	STARTING:
		FOR i := 1 TO fbCurrentSequence.stepsTotal() BY 1 DO
			Steps := fbCurrentSequence.steps();
			Steps[i].Device^.enable();
		END_FOR
		
	
		nCurrentStepPreviousCycle := nCurrentStep;
		
		// Attempt next step execution for a wait for action step
		IF Steps[nCurrentStep].WaitForAction THEN
			IF(executeStep(fbCurrentSequence.step(nCurrentStep)) AND nCurrentStep <> fbCurrentSequence.stepsTotal()) THEN
				nCurrentStep := nCurrentStep + 1;	
			END_IF
		END_IF
		
		// Attempt next step execution for a non wait for action step
		IF NOT Steps[nCurrentStep].WaitForAction THEN
			fbCurrentSequence.step(nCurrentStep)^.Device^.setCommand(StateTarget := fbCurrentSequence.step(nCurrentStep)^.Command);
			nCurrentStep := nCurrentStep + 1;	
		END_IF
		
		
		// Check which sequence step we are up to, set the currentStep indicator to +1 of where we are
		// Interlocks / permissives can cause us to go backwards in steps, therefore we must do this check
		
		IF NOT fbCurrentSequence.getSeqType() THEN // only do this check if it is a flooding sequence
			checkCurrentStep();	
			IF nCurrentStep < nCurrentStepPreviousCycle THEN  // an interlock has caused the program to roll back in sequence (interlock etc.) - stay in PAUSE state and wait for user acknowledgement
				eSMState := HOLD;
			END_IF
		END_IF
			
		eState := E_SequenceState.STARTING;
	
		
		
		
	RUNNING:


// Sequence is running - just need to check that we are still running, if not, we go to paused
		nCurrentStepPreviousCycle := nCurrentStep;
		
		IF NOT fbCurrentSequence.getSeqType() THEN // only do this check if it is a flooding sequence
			checkCurrentStep();
			IF nCurrentStep < fbCurrentSequence.stepsTotal() THEN  // something has forced us out of the running state, go to paused and wait for operator to acknowledge
				eSMState := HOLD;
			END_IF
		END_IF
		
		IF NOT (fbCurrentSequence.getSeqType()) THEN // the sequence is a floop type sequence
			eState := E_SequenceState.RUN;
		ELSIF NOT (fbCurrentSequence.step(StepNum := nCurrentStep)^.Device^.getState() = fbCurrentSequence.stepCommand(StepNumber := nCurrentStep)) THEN
			eSMState := STARTING;
		END_IF
		
		
	HOLD:
		// Do not progress the sequence until the operator has acknowledged that something went wrong
		IF bPauseAcknowledged THEN
			eSMState := STARTING;
			bPauseAcknowledged := FALSE;
		END_IF
		
		eState := E_SequenceState.HOLD;
		
	COMPLETE:
		eState := E_SequenceState.COMPLETE;
		
		
END_CASE

METHOD acknowledgePause : BOOL
VAR_INPUT
END_VAR
bPauseAcknowledged := TRUE;
END_METHOD

METHOD addSequence : BOOL
VAR_INPUT
	Sequence: FB_SequenceBase;
END_VAR
aSequences[nNumberSequences + 1] := Sequence;
nNumberSequences := nNumberSequences + 1;
END_METHOD

METHOD checkCurrentStep : BOOL
VAR_INPUT
END_VAR

VAR
	currentState: E_DeviceState;
	targetState: E_DeviceState;
END_VAR
nCurrentStepCheck := 1;

WHILE nCurrentStepCheck < (fbCurrentSequence.stepsTotal() + 1) DO
	
	currentState := fbCurrentSequence.stepState(nCurrentStepCheck);
	targetState := fbCurrentSequence.stepCommand(nCurrentStepCheck);

	IF currentState = targetState THEN
		nCurrentStepCheck := nCurrentStepCheck + 1;
	ELSE
		nCurrentStep := nCurrentStepCheck; // step check reveals we are here
		nCurrentStepCheck := fbCurrentSequence.stepsTotal() + 1; // terminate loop as the checking is finished
	END_IF
END_WHILE
END_METHOD

METHOD executeStep : BOOL
VAR_INPUT
	stSequenceStep: POINTER TO ST_SequenceStep;
END_VAR

VAR
	(*eCheckState: E_DeviceState;
	eCheckStateAlternative: E_DeviceState;
	eCheckStateAlternative2: E_DeviceState;
	eCheckCommand: E_DeviceState;
	fbDevice: POINTER TO FB_BaseDevice;
	*)
END_VAR
executeStep := FALSE;


IF fbCurrentSequence.step(StepNum := nCurrentStep)^.Device^.getState()  
	= fbCurrentSequence.stepCommand(StepNumber := nCurrentStep)
	AND fbTONstep.Q THEN  
	
	IF (nCurrentStep = fbCurrentSequence.stepsTotal() AND fbCurrentSequence.getSeqType()) THEN
		eSMState := COMPLETE;
	ELSIF (nCurrentStep = fbCurrentSequence.stepsTotal() AND (NOT fbCurrentSequence.getSeqType())) THEN
		eSMState := RUNNING;
	END_IF
	//fbTONdelay.IN := FALSE;
	fbTONdelay(IN:= TRUE, PT := stSequenceStep^.DelayUntilNextStep); 
	
	executeStep := TRUE; // indicate that the step was sucessful
	
	
ELSIF (fbCurrentSequence.step(StepNum := nCurrentStep)^.Device^.isEnabled() ) AND 
		(NOT (fbCurrentSequence.step(StepNum := nCurrentStep)^.Device^.getMode() = E_DeviceMode.MANUAL)) AND
		fbTONdelay.Q THEN 
	//AND fbTONdelay.Q THEN
		
		//fbTONdelay.IN := FALSE; 		
		fbTONdelay.IN := FALSE;
		fbTONstep(IN:= TRUE, PT := stSequenceStep^.StepMinDuration);		
		stSequenceStep^.Device^.setCommand(StateTarget := stSequenceStep^.Command); // set the target state 

END_IF

(*
IF fbCurrentSequence.step(StepNum := nCurrentStep)^.Device^.getState()  
	= fbCurrentSequence.step(StepNum := nCurrentStep)^.Device^.getCommand() 
	AND fbTONstep.Q THEN  *)
END_METHOD

METHOD getCurrentSeq_FB : POINTER TO FB_SequenceBase
VAR_INPUT
END_VAR
getCurrentSeq_FB := ADR(fbCurrentSequence);
END_METHOD

METHOD getCurrentSeq_ID : INT
VAR_INPUT
END_VAR
getCurrentSeq_ID := nCurrentSequence;
END_METHOD

METHOD getState : E_SequenceState
VAR_INPUT
END_VAR
getState := eState;
END_METHOD

METHOD initSequence : BOOL
VAR_INPUT
END_VAR
// We want to iterate through all of the components in a sequence and enable them.
// We also want to disable any other device (provided it is not in manual)
END_METHOD

METHOD pauseSequence : BOOL
VAR_INPUT
END_VAR
eSMState := HOLD;
END_METHOD

METHOD selectSequence : BOOL
VAR_INPUT
	Sequence: INT;
END_VAR
fbCurrentSequence := aSequences[Sequence];
nCurrentSequence := Sequence;
END_METHOD

METHOD startSequence : BOOL
VAR_INPUT
END_VAR
VAR

END_VAR
eSMState := STARTING;

FOR i := 1 TO fbCurrentSequence.stepsTotal() BY 1 DO
	Steps := fbCurrentSequence.steps();
	Steps[i].Device^.enable();
END_FOR

nCurrentStep := 1;
nCurrentStepPreviousCycle := 1;
//nCurrentSequence := 1;
nCurrentStepCheck := 1; 

fbTONdelay(PT := T#1s, IN := TRUE);
END_METHOD

METHOD stopSequence : BOOL
VAR_INPUT
END_VAR
eSMState := STOPPED;


FOR i := 1 TO fbCurrentSequence.stepsTotal() BY 1 DO
	Steps := fbCurrentSequence.steps();
	Steps[i].Device^.disable();
END_FOR
END_METHOD

END_FUNCTION_BLOCK

// ---- POUs/05 Sequences/FB_SequenceBase.TcPOU
(*
		This function block serves as a template for all machine sequences
		Each sequence step is a structure (ST_SequenceStep) which is defined in the FB_Init
		method of machine sequence function blocks that extend this FB.
		After the steps are defined, the STs are packed into the array 'aSequenceSteps'
		which is used by the Sequence Manager whom iterates over this array to co-ordinate 
		the execution of steps and/or detection of where sequences are interruped by interlock
		conditions
*)

FUNCTION_BLOCK FB_SequenceBase

(*
VAR_IN_OUT
	{attribute 'OPC.UA.DA' := '0'} 
	devices: ST_DMComponents;
END_VAR
*)


VAR
	sSequenceName: STRING;
	sSequenceDescription: STRING(245);
	nNumberSequenceSteps: INT;
	
	
	bSequentional_1_Flood_0: BOOL := FALSE; // default to flood and set to TRUE using setSequential() method
	
	aSequenceSteps: ARRAY[1..20] OF ST_SequenceStep;
	//aSequenceSteps: ARRAY[1..20] OF ST_SequenceStep;
	{attribute 'OPC.UA.DA' := '0'} 
	Step1: ST_SequenceStep;
	{attribute 'OPC.UA.DA' := '0'} 
	Step2: ST_SequenceStep;
	{attribute 'OPC.UA.DA' := '0'} 
	Step3: ST_SequenceStep;
	{attribute 'OPC.UA.DA' := '0'} 
	Step4: ST_SequenceStep;
	{attribute 'OPC.UA.DA' := '0'} 
	Step5: ST_SequenceStep;
	{attribute 'OPC.UA.DA' := '0'} 
	Step6: ST_SequenceStep;
	{attribute 'OPC.UA.DA' := '0'} 
	Step7: ST_SequenceStep;
	{attribute 'OPC.UA.DA' := '0'} 
	Step8: ST_SequenceStep;
	{attribute 'OPC.UA.DA' := '0'} 
	Step9: ST_SequenceStep;
	{attribute 'OPC.UA.DA' := '0'} 
	Step10: ST_SequenceStep;
	{attribute 'OPC.UA.DA' := '0'} 
	Step11: ST_SequenceStep;
	{attribute 'OPC.UA.DA' := '0'} 
	Step12: ST_SequenceStep;
	{attribute 'OPC.UA.DA' := '0'} 
	Step13: ST_SequenceStep;
	{attribute 'OPC.UA.DA' := '0'} 
	Step14: ST_SequenceStep;
	{attribute 'OPC.UA.DA' := '0'} 
	Step15: ST_SequenceStep;
	{attribute 'OPC.UA.DA' := '0'} 
	Step16: ST_SequenceStep;
	{attribute 'OPC.UA.DA' := '0'} 
	Step17: ST_SequenceStep;
	{attribute 'OPC.UA.DA' := '0'} 
	Step18: ST_SequenceStep;
	{attribute 'OPC.UA.DA' := '0'} 
	Step19: ST_SequenceStep;
	{attribute 'OPC.UA.DA' := '0'} 
	Step20: ST_SequenceStep;
	{attribute 'OPC.UA.DA' := '0'} 
	Step21: ST_SequenceStep;
	{attribute 'OPC.UA.DA' := '0'} 
	Step22: ST_SequenceStep;
	{attribute 'OPC.UA.DA' := '0'} 
	Step23: ST_SequenceStep;
	{attribute 'OPC.UA.DA' := '0'} 
	Step24: ST_SequenceStep;
	{attribute 'OPC.UA.DA' := '0'} 
	Step25: ST_SequenceStep;
	{attribute 'OPC.UA.DA' := '0'} 
	Step26: ST_SequenceStep;
	{attribute 'OPC.UA.DA' := '0'} 
	Step27: ST_SequenceStep;
	{attribute 'OPC.UA.DA' := '0'} 
	Step28: ST_SequenceStep;
END_VAR

(*
	Use the text below in the FBs that extend this to build the sequence
	
			Step1.Component := devices.
			Step1.Command := E_DeviceState.
			Step1.StepMinDuration := T#5S; 
			Step1.DelayUntilNextStep := T#5S;
			Step1.WaitForAction := TRUE;
			aSequenceSteps[1] :=   Step1;
			
			
			Step2.Component := devices.
			Step2.Command := E_DeviceState.
			Step2.StepMinDuration := T#5S; 
			Step2.DelayUntilNextStep := T#5S;
			Step2.WaitForAction := TRUE;
			aSequenceSteps[2] :=   Step2;
			
			
			Step3.Component := devices.
			Step3.Command := E_DeviceState.
			Step3.StepMinDuration := T#5S; 
			Step3.DelayUntilNextStep := T#5S;
			Step3.WaitForAction := TRUE;
			aSequenceSteps[3] :=   Step3;
			
			
			Step4.Component := devices.
			Step4.Command := E_DeviceState.
			Step4.StepMinDuration := T#5S; 
			Step4.DelayUntilNextStep := T#5S;
			Step4.WaitForAction := TRUE;
			aSequenceSteps[4] :=   Step4;
			
			
			Step5.Component := devices.
			Step5.Command := E_DeviceState.
			Step5.StepMinDuration := T#5S; 
			Step5.DelayUntilNextStep := T#5S;
			Step5.WaitForAction := TRUE;
			aSequenceSteps[5] :=   Step5;
			
			
			Step6.Component := devices.
			Step6.Command := E_DeviceState.
			Step6.StepMinDuration := T#5S; 
			Step6.DelayUntilNextStep := T#5S;
			Step6.WaitForAction := TRUE;
			aSequenceSteps[6] :=   Step6;
			
			
			Step7.Component := devices.
			Step7.Command := E_DeviceState.
			Step7.StepMinDuration := T#5S; 
			Step7.DelayUntilNextStep := T#5S;
			Step7.WaitForAction := TRUE;
			aSequenceSteps[7] :=   Step7;
			
			
			Step8.Component := devices.
			Step8.Command := E_DeviceState.
			Step8.StepMinDuration := T#5S; 
			Step8.DelayUntilNextStep := T#5S;
			Step8.WaitForAction := TRUE;
			aSequenceSteps[8] :=   Step8;
			
			
			Step9.Component := devices.
			Step9.Command := E_DeviceState.
			Step9.StepMinDuration := T#5S; 
			Step9.DelayUntilNextStep := T#5S;
			Step9.WaitForAction := TRUE;
			aSequenceSteps[9] :=   Step9;
			
			
			Step10.Component := devices.
			Step10.Command := E_DeviceState.
			Step10.StepMinDuration := T#5S; 
			Step10.DelayUntilNextStep := T#5S;
			Step10.WaitForAction := TRUE;
			aSequenceSteps[10] :=   Step10;
			
			
			Step11.Component := devices.
			Step11.Command := E_DeviceState.
			Step11.StepMinDuration := T#5S; 
			Step11.DelayUntilNextStep := T#5S;
			Step11.WaitForAction := TRUE;
			aSequenceSteps[11] :=   Step11;
			
			
			Step12.Component := devices.
			Step12.Command := E_DeviceState.
			Step12.StepMinDuration := T#5S; 
			Step12.DelayUntilNextStep := T#5S;
			Step12.WaitForAction := TRUE;
			aSequenceSteps[12] :=   Step12;
			
			
			Step13.Component := devices.
			Step13.Command := E_DeviceState.
			Step13.StepMinDuration := T#5S; 
			Step13.DelayUntilNextStep := T#5S;
			Step13.WaitForAction := TRUE;
			aSequenceSteps[13] :=   Step13;
			
			
			Step14.Component := devices.
			Step14.Command := E_DeviceState.
			Step14.StepMinDuration := T#5S; 
			Step14.DelayUntilNextStep := T#5S;
			Step14.WaitForAction := TRUE;
			aSequenceSteps[14] :=   Step14;
			
			
			Step15.Component := devices.
			Step15.Command := E_DeviceState.
			Step15.StepMinDuration := T#5S; 
			Step15.DelayUntilNextStep := T#5S;
			Step15.WaitForAction := TRUE;
			aSequenceSteps[15] :=   Step15;
			
			
			Step16.Component := devices.
			Step16.Command := E_DeviceState.
			Step16.StepMinDuration := T#5S; 
			Step16.DelayUntilNextStep := T#5S;
			Step16.WaitForAction := TRUE;
			aSequenceSteps[16] :=   Step16;
			
			
			Step17.Component := devices.
			Step17.Command := E_DeviceState.
			Step17.StepMinDuration := T#5S; 
			Step17.DelayUntilNextStep := T#5S;
			Step17.WaitForAction := TRUE;
			aSequenceSteps[17] :=   Step17;
			
			
			Step18.Component := devices.
			Step18.Command := E_DeviceState.
			Step18.StepMinDuration := T#5S; 
			Step18.DelayUntilNextStep := T#5S;
			Step18.WaitForAction := TRUE;
			aSequenceSteps[18] :=   Step18;
			
			
			Step19.Component := devices.
			Step19.Command := E_DeviceState.
			Step19.StepMinDuration := T#5S; 
			Step19.DelayUntilNextStep := T#5S;
			Step19.WaitForAction := TRUE;
			aSequenceSteps[19] :=   Step19;
			
			
			Step20.Component := devices.
			Step20.Command := E_DeviceState.
			Step20.StepMinDuration := T#5S; 
			Step20.DelayUntilNextStep := T#5S;
			Step20.WaitForAction := TRUE;
			aSequenceSteps[20] :=   Step20;



*)

METHOD getSeqType : BOOL
VAR_INPUT
END_VAR
getSeqType := bSequentional_1_Flood_0;
END_METHOD

METHOD setSeqType : BOOL
VAR_INPUT
	Sequential_1_Flood_0: BOOL;
END_VAR
bSequentional_1_Flood_0 := Sequential_1_Flood_0;
END_METHOD

METHOD step : POINTER TO ST_SequenceStep
VAR_INPUT
	StepNum: INT;
END_VAR
step := ADR(aSequenceSteps[StepNum]);
END_METHOD

METHOD stepCommand : E_DeviceState
VAR_INPUT
	StepNumber: INT;
END_VAR
stepCommand := aSequenceSteps[StepNumber].Command;
END_METHOD

METHOD steps : ARRAY[1..20] OF ST_SequenceStep
VAR_INPUT
END_VAR
steps := aSequenceSteps;
END_METHOD

METHOD stepState : E_DeviceState
VAR_INPUT
	StepNumber: INT;
END_VAR
stepState := aSequenceSteps[StepNumber].Device^.getState();
END_METHOD

METHOD stepsTotal : INT
VAR_INPUT
END_VAR
stepsTotal := nNumberSequenceSteps;
END_METHOD

METHOD updateVarIDs : BOOL
VAR
	iterator: INT;
END_VAR
FOR iterator := 1 TO nNumberSequenceSteps BY 1 DO
	aSequenceSteps[iterator].DeviceVarID := aSequenceSteps[iterator].Device^.getVarID();
END_FOR
END_METHOD

END_FUNCTION_BLOCK

// ---- POUs/00 Interfaces/FB_HandShake_TrayMovement.TcPOU
FUNCTION_BLOCK FB_HandShake_TrayMovement EXTENDS FB_BaseDevice



VAR_INPUT PERSISTENT 
	stTrayExchangeInput: ST_TrayExchangeHandshake;
END_VAR

VAR_OUTPUT PERSISTENT
	stTrayExchgangeOutput: ST_TrayExchangeHandshake;
END_VAR


VAR
	fbTON_Timer: TON;			// used to time duration from bExecuture move TRUE to both bDone booleans set to true
	{attribute 'OPC.UA.DA' := '1'} 
	tDurationMovement: TIME;	// holds the duration of the last tray movement


END_VAR

VAR PERSISTENT
	{attribute 'OPC.UA.DA' := '1'} 
	tAlarmMovement: TIME;		// user specified duration for tray movement alarm
END_VAR

fbTON_Timer(IN := (stTrayExchangeInput.eState = E_TrayExchangeState.IN_PROGRESS));

IF fbTON_Timer.Q THEN
	 aErrors[1].bEnabled 	:= TRUE;
	 aErrors[1].ePriority 	:= E_AlarmPriority.High;
	 aErrors[1].sLabel 		:= 'Tray Movement Timeout';
END_IF 

IF stTrayExchangeInput.bDoneReceiver AND stTrayExchangeInput.bDoneSender THEN
	stTrayExchangeInput.eState := E_TrayExchangeState.COMPLETED;
END_IF

IF stTrayExchangeInput.eState = E_TrayExchangeState.IN_PROGRESS THEN
	stTrayExchangeInput.stTrayOutgoing := stTrayExchangeInput.stTrayIncoming;
END_IF


stTrayExchgangeOutput := stTrayExchangeInput;

END_FUNCTION_BLOCK

// ---- POUs/LFT/FB_Lift.TcPOU
FUNCTION_BLOCK FB_Lift EXTENDS FB_BaseDevice

VAR
	fbServo: FB_SEW_MovidriveB;
END_VAR

VAR PERSISTENT
	bAbove_1_or_Below_0_HomePos: BOOL;
	bExtending_1_or_Retracting_0: BOOL;
	eSMState: (INIT, ENABLE, MOVE_TRIG, MOVING, MOVED, STOP, ERROR, RESET) := INIT;
	nGearRation: REAL; 
	nInertia: REAL;
END_VAR

END_FUNCTION_BLOCK

// ---- POUs/LFT/FB_LiftArm.TcPOU
FUNCTION_BLOCK FB_LiftArm EXTENDS FB_BaseDevice

VAR
	fbServo: FB_SEW_MovidriveB;
END_VAR
(*
VAR_IN_OUT
	fbSensor_PressSwitch: FB_AutoSwitch;
END_VAR
*)
VAR PERSISTENT
	bAbove_1_or_Below_0_HomePos: BOOL;
	bExtending_1_or_Retracting_0: BOOL;
	eSMState: (INIT, ENABLE, MOVE_TRIG, MOVING, MOVED, STOP, ERROR, RESET) := INIT;
	nGearRation: REAL; 
	nInertia: REAL;
END_VAR

END_FUNCTION_BLOCK

// ---- POUs/POP/FB_AutoSwitch.TcPOU
FUNCTION_BLOCK FB_AutoSwitch EXTENDS FB_BaseDevice
VAR
	bRawInput AT %I*: BOOL;
END_VAR

IF bRawInput THEN
	eState := E_DeviceState.ON;
ELSE
	eState := E_DeviceState.OFF;
END_IF

END_FUNCTION_BLOCK

// ---- POUs/LFT/FB_AutoGreaser.TcPOU
FUNCTION_BLOCK FB_AutoGreaser EXTENDS FB_BaseDevice
VAR_INPUT
END_VAR
VAR_OUTPUT
END_VAR
VAR
END_VAR

END_FUNCTION_BLOCK

// ---- POUs/01 Actuators/FB_Valve_ONOFF_woMonitoring.TcPOU
{attribute 'OPC.UA.DA' := '1'}
FUNCTION_BLOCK FB_Valve_ONOFF_woMonitoring EXTENDS FB_BaseDevice IMPLEMENTS I_Device, I_ValveActuated


(*
VAR_INPUT
	bNO_or_NC_0_or_1: BOOL;
END_VAR
*)

VAR
	bFirstRun: BOOL := TRUE;
	{attribute 'OPC.UA.DA' := '1'} 
	bValveOutput AT %Q*: BOOL := FALSE;
	
	{attribute 'OPC.UA.DA' := '0'} 
	eSMState: (WAIT, CLOSED, OPEN);
	
	tDebounce: TIME := T#5S;
	fbTON_Debounce: TON := (PT := tDebounce, IN := FALSE);
	
	
END_VAR

VAR PERSISTENT
	bNO_or_NC_0_or_1: BOOL; 
	bNCNC_Override: BOOL := FALSE;
END_VAR

fbTONstartTime();
fbTONstopTime();
fbTON_Debounce();

IF bFirstRun THEN
	fbTON_Debounce(IN := TRUE);
	bFirstRun := FALSE;
END_IF

IF GVL.bAutoUpdateDeviceState THEN
	eState := eStateTarget;	
END_IF

IF eMode = E_DeviceMode.MANUAL THEN
	bEnable := TRUE;
END_IF

IF (eStateTarget = E_DeviceState.OPEN) AND fbTON_Debounce.Q AND bEnable THEN
	eSMState := OPEN;
	fbTON_Debounce(IN := FALSE);
END_IF

IF eStateTarget = E_DeviceState.CLOSED OR (NOT bEnable) THEN
	eSMState := CLOSED;
	fbTON_Debounce(IN := TRUE);
END_IF

	
CASE eSMState OF
	
	WAIT:
		//Wait for method call to change ESMState
		
	OPEN:
		IF bNO_or_NC_0_or_1 THEN
			bValveOutput := TRUE;
		ELSE
			bValveOutput := FALSE;
		END_IF
		
		eState := E_DeviceState.OPEN;
		fbTON_Debounce(IN := TRUE);
	

	CLOSED:
		IF bNO_or_NC_0_or_1 THEN
			bValveOutput := FALSE;
		ELSE
			bValveOutput := TRUE;
		END_IF
		
		eState := E_DeviceState.CLOSED;
		fbTON_Debounce(IN := TRUE);
END_CASE

{warning 'add method implementation '}
METHOD close : BOOL
IF bEnable = TRUE THEN
	eStateTarget := E_DeviceState.CLOSED;
END_IF
END_METHOD

{warning 'add method implementation '}
METHOD disable : BOOL
bEnable := FALSE;
END_METHOD

{warning 'add method implementation '}
METHOD enable : BOOL
bEnable := TRUE;
END_METHOD

{warning 'add method implementation '}
METHOD FB_init : BOOL
VAR_INPUT
	(* if TRUE, the retain variables are initialized (warm start / cold start)*)
	bInitRetains	: BOOL;
	(* if TRUE, the instance afterwards gets moved into the copy code (online change)*)
	bInCopyCode	: BOOL;
	
	ValveID: STRING(80);
	ValveDescr: STRING(255); 
	
	Normal_State_NC_1_NO_0: BOOL;
END_VAR
sID := ValveID;
sDescr := ValveDescr;

bNO_or_NC_0_or_1 := Normal_State_NC_1_NO_0;
END_METHOD

METHOD getMode : E_DeviceMode
VAR_INPUT
END_VAR

getMode := eMode;
END_METHOD

{warning 'add method implementation '}
METHOD open : BOOL
IF bEnable = TRUE THEN
	eStateTarget := E_DeviceState.OPEN;
END_IF
END_METHOD

END_FUNCTION_BLOCK

// ---- POUs/99 Utilities/FB_InterlockManager.TcPOU
FUNCTION_BLOCK FB_InterlockManager

VAR
	aInterlocks: ARRAY[1..50] OF ST_Interlock;
	nIterator: INT := 1;
END_VAR

METHOD execute : BOOL
VAR_INPUT
END_VAR

VAR
	iterator: INT;

	
	Active:			BOOL;
	Bridge:			BOOL;
	SubjectDevice:	POINTER TO FB_BaseDevice;
	SubjectState:	E_DeviceState;
	Signal:			BOOL;
	Description: 	STRING(255);
	HoldSeq:		BOOL;
	InterlockType:	E_InterlockType;
	
	
	
END_VAR

FOR iterator:=1 TO nIterator BY 1 DO
	
	// Update local variable on each loop iteration
	
	Active := aInterlocks[iterator].Active;
	Bridge := aInterlocks[iterator].Bridge;
	SubjectDevice := aInterlocks[iterator].SubjectDevice;
	SubjectState  := aInterlocks[iterator].SubjectState;
	Signal := aInterlocks[iterator].Signal;
	HoldSeq := aInterlocks[iterator].HoldSeq;
	InterlockType := aInterlocks[iterator].InterlockType;
	
	
	IF Signal = TRUE THEN
		
		// Interlock causes the sequence to go into hold (by disabling device)
		// Sequence hold requires operator acknowledgement to resume
		IF  SubjectDevice^.isEnabled() AND HoldSeq AND Bridge <> TRUE THEN
			
			SubjectDevice^.setCommand(StateTarget := SubjectState);
			SubjectDevice^.disable();
			aInterlocks[iterator].Active := TRUE;
		
			
		// Interlock causes device to change state only
		// No operator acknowledgement required 
		ELSIF  SubjectDevice^.isEnabled() AND HoldSeq =FALSE AND Bridge <> TRUE THEN
			
			SubjectDevice^.setCommand(StateTarget := SubjectState);
			aInterlocks[iterator].Active := TRUE;
			
		ELSE
			aInterlocks[iterator].Active := FALSE;
		END_IF
		
	ELSE
		aInterlocks[iterator].Active := FALSE;
	END_IF
END_FOR
END_METHOD

METHOD init : BOOL
VAR_INPUT
END_VAR
// Reset the iterator on each cycle of the machine
nIterator := 1;
END_METHOD

METHOD update : BOOL
VAR_INPUT
	Description:	STRING;
	InterlockType: 	E_InterlockType;
	Subject_Device: POINTER TO FB_BaseDevice;
	Subject_State:	E_DeviceState;
	Signal: 		BOOL;
	HoldSequence: 	BOOL;
END_VAR
aInterlocks[nIterator].HoldSeq := HoldSequence;
aInterlocks[nIterator].InterlockType := InterlockType;
aInterlocks[nIterator].Signal := Signal;
aInterlocks[nIterator].Description := Description;
aInterlocks[nIterator].SubjectDevice := Subject_Device;
aInterlocks[nIterator].SubjectVarID := Subject_Device^.getVarID();
aInterlocks[nIterator].SubjectState := Subject_State;

nIterator := nIterator + 1;
END_METHOD

END_FUNCTION_BLOCK

// ---- POUs/00 Interfaces/FB_BaseMachine_1.TcPOU
{attribute 'OPC.UA.DA.StructuredType' := '1'}
FUNCTION_BLOCK FB_BaseMachine_1
VAR

	{attribute 'OPC.UA.DA' := '0'} 
	bBusy: BOOL := FALSE;
	{attribute 'OPC.UA.DA' := '1'} 
	bError: BOOL := FALSE;
	{attribute 'OPC.UA.DA' := '1'} 
	bEnable: BOOL := FALSE;
	{attribute 'OPC.UA.DA' := '1'} 
	eState: E_MachineState := E_MachineState.IDLE;
	{attribute 'OPC.UA.DA' := '1'} 
	{attribute 'OPC.UA.DA.StructuredType' := '1'}
	fbSequenceManager: FB_SequenceManager_1;
	{attribute 'OPC.UA.DA' := '0'} 
	aAllComponents: ARRAY[1..50] OF POINTER TO FB_BaseDevice;
	
	{attribute 'OPC.UA.DA' := '1'} 
	aErrors: ARRAY[1..20] OF ST_Alarm;	// raiseEvent() method updates Error1 / aErrors[1] only at the moment, must implement a ring buffer with error active checking for full functionality

	
END_VAR 

VAR_INPUT
	{attribute 'OPC.UA.DA' := '1'} 
	sID: STRING;  
	{attribute 'OPC.UA.DA' := '1'} 
	sDescr: STRING;
	{attribute 'OPC.UA.DA' := '1'} 
	nQtyComponents: INT;
END_VAR

METHOD devices_disable_All : BOOL
VAR
	iterator: INT;
	
END_VAR
FOR iterator:=1 TO nQtyComponents BY 1 DO
	aAllComponents[iterator]^.disable();
END_FOR
END_METHOD

METHOD devices_disable_CurrSeq : BOOL
VAR
	iterator: INT;
	Steps : ARRAY[1..20] OF ST_SequenceStep;
END_VAR
FOR iterator:=1 TO fbSequenceManager.getCurrentSeq_FB()^.stepsTotal() BY 1 DO
	
	Steps := fbSequenceManager.getCurrentSeq_FB()^.steps();
	Steps[iterator].Device^.disable();
	
END_FOR
END_METHOD

METHOD devices_enable_All : BOOL
VAR
	iterator: INT;
END_VAR
FOR iterator:=1 TO nQtyComponents BY 1 DO
	aAllComponents[iterator]^.enable();
END_FOR
END_METHOD

METHOD devices_enable_CurrSeq : BOOL
VAR
	iterator: INT;
	Steps : ARRAY[1..20] OF ST_SequenceStep;
END_VAR
FOR iterator:=1 TO fbSequenceManager.getCurrentSeq_FB()^.stepsTotal() BY 1 DO
	Steps := fbSequenceManager.getCurrentSeq_FB()^.steps();
	Steps[iterator].Device^.enable();
END_FOR
END_METHOD

METHOD devices_setAuto_All : BOOL
VAR
	iterator: INT;
END_VAR
FOR iterator:=1 TO nQtyComponents BY 1 DO
	aAllComponents[iterator]^.setMode(Mode := E_DeviceMode.AUTO);
END_FOR
END_METHOD

METHOD devices_setAuto_CurrSeq : BOOL
VAR
	iterator: INT;
	Steps : ARRAY[1..20] OF ST_SequenceStep;
END_VAR
FOR iterator:=1 TO fbSequenceManager.getCurrentSeq_FB()^.stepsTotal() BY 1 DO
	
	Steps := fbSequenceManager.getCurrentSeq_FB()^.steps();
	Steps[iterator].Device^.setMode(Mode := E_DeviceMode.AUTO);
END_FOR
END_METHOD

METHOD devices_setManual_All : BOOL
VAR
	iterator: INT;
END_VAR
FOR iterator:=1 TO nQtyComponents BY 1 DO
	aAllComponents[iterator]^.setMode(Mode := E_DeviceMode.AUTO);
END_FOR
END_METHOD

METHOD devices_setManual_CurrSeq : BOOL
VAR
	iterator: INT;
	Steps : ARRAY[1..20] OF ST_SequenceStep;
END_VAR
FOR iterator:=1 TO fbSequenceManager.getCurrentSeq_FB()^.stepsTotal() BY 1 DO
	
	Steps := fbSequenceManager.getCurrentSeq_FB()^.steps();
	Steps[iterator].Device^.setMode(Mode := E_DeviceMode.MANUAL);
END_FOR
END_METHOD

METHOD seq_Pause : BOOL
VAR_INPUT
END_VAR
fbSequenceManager.pauseSequence();
END_METHOD

METHOD seq_Start : BOOL
VAR_INPUT
	SeqNum: UINT;
END_VAR
devices_disable_All();
fbSequenceManager.selectSequence(Sequence := 1);
devices_enable_CurrSeq();
fbSequenceManager.startSequence();
END_METHOD

METHOD seq_Stop : BOOL
VAR_INPUT
END_VAR
fbSequenceManager.stopSequence();
END_METHOD

END_FUNCTION_BLOCK

// ---- POUs/05 Sequences/FB_SequenceManager_1.TcPOU
(*
		The sequence manager co-ordinates the selection and execution of 
		machine sequences. Machine sequences are created by extending the 
		FB_SequenceBase FB.
*)

FUNCTION_BLOCK FB_SequenceManager_1
VAR	
	//aSequences: ARRAY[1..5] OF POINTER TO FB_SequenceBase;
	 
	nNumberSequences: INT := 0;
	
	{attribute 'OPC.UA.DA' := '1'} 
	eState:  E_SequenceState := E_SequenceState.STOP; //always stop sequences after PLC restart
	{attribute 'OPC.UA.DA' := '1'} 
	eStateTarget:  E_SequenceState := E_SequenceState.STOP;
	
	eSMState: (STOPPED, STARTING, RUNNING, HOLD) := STOPPED;
	nCurrentStep: INT := 1;
	nCurrentStepPreviousCycle: INT := 1;
	nCurrentSequence: INT := 1;
	nCurrentStepCheck: INT := 1; // use this to iterate over the sequence steps to check if an interlock has rolled back the sequence
	bPauseAcknowledged: BOOL := FALSE;
	
	{attribute 'OPC.UA.DA' := '0'} 
	fbTONstep: TON;			// these timers are set using the time values stored in each ST_SequenceStep
	{attribute 'OPC.UA.DA' := '0'} 
	fbTONdelay: TON;
	{attribute 'OPC.UA.DA' := '0'} 
	bIsFirstRun: BOOL := TRUE;
	
	i: INT;
	Steps : ARRAY[1..20] OF ST_SequenceStep;
	
	fbCurrentSequence: FB_SequenceBase;
END_VAR

VAR_IN_OUT
	aSequences: ARRAY[1..10] OF FB_SequenceBase;
	//fbCurrentSequence: FB_SequenceBase;
END_VAR

IF bIsFirstRun THEN
	fbTONdelay.PT := T#0S;
	fbTONdelay.IN := TRUE;
	fbTONdelay.PT := T#0S;
	fbTONstep.IN := FALSE;
	bIsFirstRun := FALSE;
	fbCurrentSequence := aSequences[1];
	eSMState := STOPPED;
END_IF

fbTONstep();
fbTONdelay();

CASE eSMState OF
	
	STOPPED:
		// Wait here until a start sequence command is received
		eState := E_SequenceState.STOP;
		
	STARTING:
		FOR i := 1 TO fbCurrentSequence.stepsTotal() BY 1 DO
			Steps := fbCurrentSequence.steps();
			Steps[i].Device^.enable();
		END_FOR
	
		nCurrentStepPreviousCycle := nCurrentStep;
		
		// Attempt next step execution 
		IF executeStep(fbCurrentSequence.step(nCurrentStep)) AND nCurrentStep <> fbCurrentSequence.stepsTotal() THEN
			nCurrentStep := nCurrentStep + 1;
		END_IF
		
		
		// Check which sequence step we are up to, set the currentStep indicator to +1 of where we are
		// Interlocks / permissives can cause us to go backwards in steps, therefore we must do this check
		
		IF NOT fbCurrentSequence.getSeqType() THEN // only do this check if it is a flooding sequence
			checkCurrentStep();	
			IF nCurrentStep < nCurrentStepPreviousCycle THEN  // an interlock has caused the program to roll back in sequence (interlock etc.) - stay in PAUSE state and wait for user acknowledgement
				eSMState := HOLD;
			END_IF
		END_IF
			
		IF nCurrentStep = fbCurrentSequence.stepsTotal() THEN  // check if we have completed all of the steps
			eSMState := RUNNING;
		END_IF
		
		eState := E_SequenceState.STARTING;
	
		
		
		
	RUNNING:
		// Sequence is running - just need to check that we are still running, if not, we go to paused
		nCurrentStepPreviousCycle := nCurrentStep;
		
		IF NOT fbCurrentSequence.getSeqType() THEN // only do this check if it is a flooding sequence
			checkCurrentStep();
			IF nCurrentStep < fbCurrentSequence.stepsTotal() THEN  // something has forced us out of the running state, go to paused and wait for operator to acknowledge
				eSMState := HOLD;
			END_IF
		END_IF
		
		IF NOT (fbCurrentSequence.getSeqType()) THEN // the sequence is a floop type sequence
			eState := E_SequenceState.RUN;
		ELSIF fbCurrentSequence.getSeqType() AND fbTONstep.Q THEN
			eState := E_SequenceState.COMPLETE; // mark the sequential sequence as complete if it has completed the final step
		END_IF
		
		
		IF NOT (fbCurrentSequence.step(StepNum := nCurrentStep)^.Device^.getState() = fbCurrentSequence.stepCommand(StepNumber := nCurrentStep)) THEN
			eSMState := STARTING;
		END_IF
		
	HOLD:
		// Do not progress the sequence until the operator has acknowledged that something went wrong
		IF bPauseAcknowledged THEN
			eSMState := STARTING;
			bPauseAcknowledged := FALSE;
		END_IF
		
		eState := E_SequenceState.HOLD;
		
		
END_CASE

METHOD acknowledgePause : BOOL
VAR_INPUT
END_VAR
bPauseAcknowledged := TRUE;
END_METHOD

METHOD addSequence : BOOL
VAR_INPUT
	Sequence: FB_SequenceBase;
END_VAR
aSequences[nNumberSequences + 1] := Sequence;
nNumberSequences := nNumberSequences + 1;
END_METHOD

METHOD checkCurrentStep : BOOL
VAR_INPUT
END_VAR

VAR
	currentState: E_DeviceState;
	targetState: E_DeviceState;
END_VAR
nCurrentStepCheck := 1;

WHILE nCurrentStepCheck < (fbCurrentSequence.stepsTotal() + 1) DO
	
	currentState := fbCurrentSequence.stepState(nCurrentStepCheck);
	targetState := fbCurrentSequence.stepCommand(nCurrentStepCheck);

	IF currentState = targetState THEN
		nCurrentStepCheck := nCurrentStepCheck + 1;
	ELSE
		nCurrentStep := nCurrentStepCheck; // step check reveals we are here
		nCurrentStepCheck := fbCurrentSequence.stepsTotal() + 1; // terminate loop as the checking is finished
	END_IF
END_WHILE
END_METHOD

METHOD executeStep : BOOL
VAR_INPUT
	stSequenceStep: POINTER TO ST_SequenceStep;
END_VAR

VAR
	(*eCheckState: E_DeviceState;
	eCheckStateAlternative: E_DeviceState;
	eCheckStateAlternative2: E_DeviceState;
	eCheckCommand: E_DeviceState;
	fbDevice: POINTER TO FB_BaseDevice;
	*)
END_VAR
executeStep := FALSE;
	
// IF fbCurrentSequence.step(StepNum := nCurrentStep)^.Device^.isEnabled()  THEN 
IF (fbCurrentSequence.step(StepNum := nCurrentStep)^.Device^.isEnabled() ) AND 
		(NOT (fbCurrentSequence.step(StepNum := nCurrentStep)^.Device^.getMode() = E_DeviceMode.MANUAL)) THEN 
	//AND fbTONdelay.Q THEN
		
		//fbTONdelay.IN := FALSE; 		
		fbTONstep(IN:= TRUE, PT := stSequenceStep^.StepMinDuration);		
		stSequenceStep^.Device^.setCommand(StateTarget := stSequenceStep^.Command); // set the target state 

END_IF

(*
IF fbCurrentSequence.step(StepNum := nCurrentStep)^.Device^.getState()  
	= fbCurrentSequence.step(StepNum := nCurrentStep)^.Device^.getCommand() 
	AND fbTONstep.Q THEN  *)


IF fbCurrentSequence.step(StepNum := nCurrentStep)^.Device^.getState()  
	= fbCurrentSequence.stepCommand(StepNumber := nCurrentStep)
	AND fbTONstep.Q THEN  
	
	fbTONstep.IN := FALSE; 
	fbTONdelay.IN := FALSE;
	fbTONdelay(IN:= TRUE, PT := stSequenceStep^.DelayUntilNextStep); 
	
	executeStep := TRUE; // indicate that the step was sucessful
	
END_IF
END_METHOD

METHOD getCurrentSeq_FB : POINTER TO FB_SequenceBase
VAR_INPUT
END_VAR
getCurrentSeq_FB := ADR(fbCurrentSequence);
END_METHOD

METHOD getCurrentSeq_ID : INT
VAR_INPUT
END_VAR
getCurrentSeq_ID := nCurrentSequence;
END_METHOD

METHOD getState : E_SequenceState
VAR_INPUT
END_VAR
getState := eState;
END_METHOD

METHOD initSequence : BOOL
VAR_INPUT
END_VAR
// We want to iterate through all of the components in a sequence and enable them.
// We also want to disable any other device (provided it is not in manual)
END_METHOD

METHOD pauseSequence : BOOL
VAR_INPUT
END_VAR
eSMState := HOLD;
END_METHOD

METHOD selectSequence : BOOL
VAR_INPUT
	Sequence: INT;
END_VAR
fbCurrentSequence := aSequences[Sequence];
nCurrentSequence := Sequence;
END_METHOD

METHOD startSequence : BOOL
VAR_INPUT
END_VAR
VAR

END_VAR
eSMState := STARTING;

FOR i := 1 TO fbCurrentSequence.stepsTotal() BY 1 DO
	Steps := fbCurrentSequence.steps();
	Steps[i].Device^.enable();
END_FOR

nCurrentStep := 1;
nCurrentStepPreviousCycle := 1;
//nCurrentSequence := 1;
nCurrentStepCheck := 1;
END_METHOD

METHOD stopSequence : BOOL
VAR_INPUT
END_VAR
eSMState := STOPPED;


FOR i := 1 TO fbCurrentSequence.stepsTotal() BY 1 DO
	Steps := fbCurrentSequence.steps();
	Steps[i].Device^.disable();
END_FOR
END_METHOD

END_FUNCTION_BLOCK

// ---- POUs/00 Interfaces/FB_BaseSensor.TcPOU
{attribute 'OPC.UA.DA.StructuredType' := '1'}
FUNCTION_BLOCK FB_BaseSensor EXTENDS FB_BaseDevice

VAR
	
	// Base Sensor Variables 
	{attribute 'OPC.UA.DA' := '0'} 
	eSensorType: E_SensorType;
	{attribute 'OPC.UA.DA' := '0'} 
	nRawInput AT %I*: INT;				// Link to IO
	{attribute 'OPC.UA.DA' := '1'} 
	nMeasuredCurrent: REAL;				// Raw-input converted to mA units
	{attribute 'OPC.UA.DA' := '1'}
	nFilteredCurrent: REAL; 			// MA filter to mA reading
	{attribute 'OPC.UA.DA' := '1'}
	nCurrentValue: REAL; 				// Unfiltered value after conversion to desired units
	{attribute 'OPC.UA.DA' := '1'}
	nCurrentValueFiltered: REAL; 		// MA & threshhold filtered after conversion to desired units
	
	
	// MA Filter Variables

	bResetTimer: 					BOOL := FALSE;
	fbTON_Filter:	 				TON := (PT := nSampleRate, IN := TRUE);
	fbFilter:						FB_SigCond_MovingAverage := (nSamplesToFilter := nQtySamples, tCtrlCycleTime := nSampleRate, tTaskCycleTime := GVL.tPLCTaskTime);
	
	
END_VAR

VAR PERSISTENT
	// MA Filter Variables
	nQtySamples:					UINT := 200;
	nSampleRate: 					TIME := T#100MS;
	
	// Threshold filtering variables
	nThresholdMin: REAL := 0;
	nThresholdMax: REAL := 1000000;
	bThresholdEnable: BOOL := FALSE;

	
END_VAR

// This is the base class for all devices (actuators and sensors)
// Provides common variables to all instances 
// Note that the I_Device interface provides the common methods for all devices

METHOD filter : BOOL
VAR_INPUT
END_VAR
IF bResetTimer THEN
	fbTON_Filter(IN := TRUE);
	bResetTimer := FALSE;
END_IF

fbTON_Filter();
fbFilter(nSamplesToFilter := nQtySamples, tCtrlCycleTime := nSampleRate, tTaskCycleTime := GVL.tPLCTaskTime);

IF fbTON_Filter.Q THEN
	fbFilter(fIn := nMeasuredCurrent);
	fbTON_Filter(IN := FALSE);
	bResetTimer := TRUE;
	nFilteredCurrent := fbFilter.fOut;
END_IF
END_METHOD

END_FUNCTION_BLOCK

// ---- POUs/97 Signal Conditioning/FB_SigCond_MovingAverage.TcPOU
FUNCTION_BLOCK FB_SigCond_MovingAverage
VAR_INPUT
	fIn:					FLOAT;
	nSamplesToFilter:		UINT; // Maximum of 500
	tCtrlCycleTime:			TIME;
	tTaskCycleTime:			TIME;

	fManSyncValue:	FLOAT;
	bSync:			BOOL;
	eMode:			E_CTRL_MODE;
	bHold:			BOOL;
END_VAR

VAR
	
	fbCtr_MovAvg:	FB_CTRL_MOVING_AVERAGE;
	stParams:		ST_CTRL_MOVING_AVERAGE_PARAMS;
	aInternalData:	ARRAY[1..500] OF FLOAT;
END_VAR


VAR_OUTPUT
	fOut:			FLOAT;
	eState:			E_CTRL_STATE;
	eErrorID:		E_CTRL_ERRORCODES;
	bError:			BOOL;	
END_VAR



// Read inputs and put into params structure
stParams.nSamplesToFilter 	:= nSamplesToFilter;
stParams.tCtrlCycleTime 	:= tCtrlCycleTime;
stParams.tTaskCycleTime		:= tTaskCycleTime;
stParams.pWorkArray_ADR		:= ADR(aInternalData);
stParams.nWorkArray_SIZEOF	:= SIZEOF(aInternalData);

eMode := E_CTRL_MODE.eCTRL_MODE_ACTIVE;

// Execute filter
fbCtr_MovAvg(fIn := fIn, fManSyncValue := fManSyncValue, bSync := bSync, eMode := eMode, bHold := bHold, stParams := stParams);


// Update outputs
fOut 		:= fbCtr_MovAvg.fOut;
eState 		:= fbCtr_MovAvg.eState;
eErrorID 	:= fbCtr_MovAvg.eErrorId;
bError 		:= fbCtr_MovAvg.bError;

END_FUNCTION_BLOCK

// ---- POUs/01 Actuators/Dosing Machine/FB_AutoClean_Filter_Bollfilter.TcPOU
FUNCTION_BLOCK FB_AutoClean_Filter_Bollfilter EXTENDS FB_BaseDevice IMPLEMENTS I_Device
VAR_INPUT
END_VAR
VAR_OUTPUT
END_VAR
VAR
END_VAR

END_FUNCTION_BLOCK

// ---- POUs/01 Actuators/Dosing Machine/FB_DosingPumpAgrowtek_R2.TcPOU
{attribute 'OPC.UA.DA.StructuredType' := '1'}
FUNCTION_BLOCK FB_DosingPumpAgrowtek_R2 EXTENDS FB_BaseDevice IMPLEMENTS I_PumpDosing

VAR_IN_OUT
	{attribute 'OPC.UA.DA' := '0'}
	//fbModbusMaster: FB_ModbusMaster;
	fbModbusManager: FB_ModbusManager;
END_VAR

VAR_INPUT
	nModbusUnitID: UINT; 
END_VAR

VAR
	// Modbus Variables
	nPumpID: UINT;	// Pump ID is different to the modbus ID because there are 5 pumps on the 1 modbus address
	 
	ePumpType: E_DosingPump;
	
	bInitialDose: BOOL;
	
	bEnableComms: BOOL := TRUE;
	bFirtRun: BOOL := TRUE;
	bResetTimer: BOOL := TRUE;
	
	// Async Statemachine Variables
	{attribute 'OPC.UA.DA' := '0'}
	eSMState: (WAIT, DOSING_TRIG, DOSING, DOSING_OFF_TRIG, DOSED);
	
	// Dosing Variables
	{attribute 'OPC.UA.DA' := '0'} 
	fbTONdoseTime: TON;  
	{attribute 'OPC.UA.DA' := '1'} 
	nDoseRateMLph: UINT;
	{attribute 'OPC.UA.DA' := '1'} 
	nDoseQtyMls: REAL;
	{attribute 'OPC.UA.DA' := '1'} 
	tTimeToDose: TIME;
	
	// delay between writing pump speed and reading pump speed
	fbTONreadDelay : TON := (PT := T#1S);

	// Variables updated over Modbus
	{attribute 'OPC.UA.DA' := '1'} 
	nPumpSpeed_Requested: UINT;
	
	{attribute 'OPC.UA.DA' := '1'} 
	nPumpSpeed: UINT;
	{attribute 'OPC.UA.DA' := '1'} 
	nPumpRunTime: UINT; 
	
	tDataRefresh: TIME := T#10S;
	fbTON_DataRefresh: 	TON := (PT := tDataRefresh, IN := FALSE);
	fbTON_MsgTimeout: 	TON := (PT := T#4S, IN := FALSE);
	
	// Modbus Requests
	stModRead_MotorSpeed: 	ST_Modbus_ReadRequest;
	stModRead_MotorRunTime: ST_Modbus_ReadRequest;
	stModWrite_MotorSpeed: 	ST_Modbus_WriteRequest;
	stModWrite_SetID: 		ST_Modbus_WriteRequest;
	
	
	bRaiseError1: BOOL := FALSE;
	bClearError: BOOL := FALSE;
	bRaiseError2: BOOL := FALSE;
	
	
END_VAR

fbTONdoseTime();
fbTON_MsgTimeout();
fbTON_DataRefresh();
fbTONreadDelay();

IF GVL.bAutoUpdateDeviceState THEN
	eState := eStateTarget;	
END_IF

IF bFirtRun THEN
	init_ModbusRequests();
	bFirtRun := FALSE;
END_IF

IF eMode = E_DeviceMode.MANUAL THEN
	bEnable := TRUE;
END_IF
(*

IF bEnable AND eStateTarget = E_DeviceState.ON AND eState <> E_DeviceState.RUNNING THEN
		eSMState := WAIT;
END_IF

IF (bEnable = FALSE OR eStateTarget = E_DeviceState.IDLE) AND eState <> E_DeviceState.IDLE THEN
		eSMState := 0;
END_IF
*)


IF bResetTimer THEN
	fbTON_DataRefresh.IN := TRUE;
	bResetTimer := FALSE;
END_IF

// Asynchronous update of local variables from the Modbus request structures
nPumpSpeed 		:= WORD_TO_UINT(stModRead_MotorSpeed.ReadRegsVals[1]);
nPumpRunTime 	:= WORD_TO_UINT(stModRead_MotorRunTime.ReadRegsVals[1]);
	
// Request update of local veriables every Xs (in accordance with adjustable DataRefresh timer)
(*IF fbTON_DataRefresh.Q AND bEnable THEN // AND bEnableComms THEN
	// fbModbusManager.addRequest_Read_Priority(ReadRequest := ADR(stModRead_MotorRunTime));
	fbModbusManager.addRequest_Read_Priority(ReadRequest := ADR(stModRead_MotorSpeed));
	fbTON_DataRefresh.IN := FALSE;
	bResetTimer := TRUE;
END_IF
*)


// Statemachine to handle dosing commands
//IF eState = E_Devicestate.RUNNING THEN //AND bEnableComms THEN
	CASE eSMState OF
	
		WAIT:
			// Wait for a dosing command
			eState := E_DeviceState.IDLE;
			// Beau make sure the timeout timer is cleared in case it was left on last time
			fbTON_MsgTimeout.IN := FALSE;
			
		DOSING_TRIG:
			// A call to the 'executeDose' has been received, send modbus command
			// Send the dosing modbus request and start the timer
			//nPumpSpeed_Requested := 100;
			stModWrite_MotorSpeed.WriteRegVals[1] := UINT_TO_WORD(nPumpSpeed_Requested);
			fbModbusManager.addRequest_Write_Priority(WriteRequest := ADR(stModWrite_MotorSpeed));
			// Beau instead of reading pump speed immediately, start the delay timer
			fbTONreadDelay.IN := TRUE;
			//fbModbusManager.addRequest_Read_Priority(ReadRequest := ADR(stModRead_MotorSpeed));
			fbTONdoseTime.IN := TRUE;
			fbTON_MsgTimeout.PT := fbTONdoseTime.PT + T#1S;
			fbTON_MsgTimeout.IN := TRUE;
			eSMState := DOSING;
			eState := E_DeviceState.RUNNING;
			
	
		DOSING: 
		
			// Beau try to read pump speed one second after writing pump speed
			IF fbTONreadDelay.Q THEN
				fbModbusManager.addRequest_Read_Priority(ReadRequest := ADR(stModRead_MotorSpeed));	
				// reset the timer so we don't send another read request
				fbTONreadDelay.IN := FALSE;
			END_IF
			
			IF fbTON_MsgTimeout.Q AND NOT (nPumpSpeed_Requested = nPumpSpeed) THEN
				// The pump hasn't turned on after it was requested to - try again!
				fbModbusManager.addRequest_Read_Priority(ReadRequest := ADR(stModRead_MotorSpeed));
				fbTONdoseTime.IN := FALSE;
				fbTON_MsgTimeout.IN := FALSE;
				eSMState := DOSING_TRIG; // go back and retry
			END_IF
			
			
			IF fbTONdoseTime.Q THEN
				fbTONdoseTime.IN := FALSE; // reset the timer
				IF nPumpSpeed = nPumpSpeed_Requested THEN
					fbTONdoseTime.IN := FALSE;
					fbTON_MsgTimeout.IN := FALSE;
					eSMState := DOSING_OFF_TRIG; // the pump turned on, now we can turn off
				END_IF
			END_IF
			eState := E_DeviceState.RUNNING;
				
			
		DOSING_OFF_TRIG:
			
			// Monitor the run time / compare against the calculated dosing time
			// when dosing time has been exceeded move to dosed
			nPumpSpeed_Requested := 0; // turn the pump off
			stModWrite_MotorSpeed.WriteRegVals[1] := UINT_TO_WORD(nPumpSpeed_Requested);
			
			fbModbusManager.addRequest_Write_Priority(WriteRequest := ADR(stModWrite_MotorSpeed));
			
			fbModbusManager.addRequest_Read_Priority(ReadRequest := ADR(stModRead_MotorSpeed));
			
			fbModbusManager.addRequest_Write_Priority(WriteRequest := ADR(stModWrite_MotorSpeed));
			fbModbusManager.addRequest_Write_Priority(WriteRequest := ADR(stModWrite_MotorSpeed));
			fbModbusManager.addRequest_Write_Priority(WriteRequest := ADR(stModWrite_MotorSpeed));
			fbTON_MsgTimeout.IN := TRUE;
			fbTON_MsgTimeout.PT := T#1s;;
			eSMState := DOSED;
			eState := E_DeviceState.RUNNING;
			
			
		DOSED: 
			// Confirm that the pump has stopped by reading the pump speed 
			// go back to wait if the pump speed has reached 0
			
			IF fbTON_MsgTimeout.Q THEN
				fbTON_MsgTimeout.IN := FALSE;
				IF NOT(nPumpSpeed_Requested = nPumpSpeed) THEN
					// The pump hasn't turned off after it was requested to - try again!
					eSMState := DOSING_OFF_TRIG; // go back and retry
				ELSIF nPumpSpeed_Requested = nPumpSpeed THEN
					eSMState := WAIT; // go back to waiting for the next dose
					nDoseQtyMls := 0; // reset this to 0 for SCADA 
				END_IF
			END_IF
			
			// eSMState := WAIT;
			
	
	END_CASE

//END_IF

{warning 'add method implementation '}
METHOD executeDose : BOOL
VAR_INPUT
	DoseQtyMls: LREAL;
	DoseRateMlph: UINT;
	RequestComplete: 	POINTER TO BOOL;
END_VAR
VAR_OUTPUT
	RequestAccepted: BOOL;
END_VAR
(* setDose dispenses the amount requested at a user requested dose rate *)

//nDoseQtyMls := REAL_TO_UINT((UINT_TO_REAL(DoseQtyMls)/10000.0));
IF (bEnable AND bEnableComms) OR (eMode = E_DeviceMode.MANUAL)  THEN
	// nDoseQtyMls := ABS(DoseQtyMls);

	// IF nDoseQtyMls > 1.0 THEN
	
		nPumpSpeed_Requested := 40;
		//tTimeToDose := REAL_TO_TIME(( nDoseQtyMls / (480.0*(UINT_TO_REAL(nPumpSpeed_Requested)/100.0))) * 60.0 *1000.0);  // Agrowtek maximum flow rate is 480 ml/min
		tTimeToDose := REAL_TO_TIME(( ABS(DoseQtyMls) / (480.0*(UINT_TO_REAL(nPumpSpeed_Requested)/100.0))) * 60.0 *1000.0);  // Agrowtek maximum flow rate is 480 ml/min
		//tTimeToDose := REAL_TO_TIME((((UINT_TO_REAL(nDoseQtyMls)) / 480) * 60.0)*1000);  // Agrowtek maximum flow rate is 480 ml/min
		fbTONdoseTime.PT := tTimeToDose;
	
		IF tTimeToDose > T#1.6S THEN
			nDoseQtyMls := ABS(DoseQtyMls);
			eSMState := DOSING_TRIG;
			eState := E_Devicestate.RUNNING;
			bBusy := TRUE;	
		END_IF
	END_IF
END_METHOD

METHOD FB_init : BOOL


VAR_INPUT
	bInitRetains : BOOL; // if TRUE, the retain variables are initialized (warm start / cold start)
	bInCopyCode : BOOL;  // if TRUE, the instance afterwards gets moved into the copy code (online change)
	
	PumpID: STRING;
	PumpDescription: STRING;
	PumpType: E_DosingPump;
	ManifoldModbusID: UINT; 
	
END_VAR
sID := PumpID;
sDescr := PumpDescription;
ePumpType := PumpType;
nModbusUnitID := ManifoldModbusID;
END_METHOD

METHOD getAdrReadAccumRunTime : UINT
VAR_INPUT
	PumpType: E_DosingPump;
END_VAR

VAR
	Address: UINT;
END_VAR
// This method retrieves the Modbus register for the individual Agrowtek pump
// We need to do this because 5 pumps share the same Modbus slave ID, however have differing registers to write to

CASE PumpType OF
	
	E_DosingPump.PH_DOWN:
		Address := 16#64;
		
	E_DosingPump.NUTRIENT_A:
		Address := 16#65;
		
	E_DosingPump.NUTRIENT_B:
		Address := 16#66;

	E_DosingPump.NUTRIENT_C:
		Address := 16#67;
		
	E_DosingPump.PH_UP:
		Address := 16#68;
		
END_CASE

getAdrReadAccumRunTime := Address;
END_METHOD

METHOD getAdrReadWriteSpeed : UINT
VAR_INPUT
	PumpType: E_DosingPump;
END_VAR
// This method retrieves the Modbus register for the individual Agrowtek pump
// We need to do this because 5 pumps share the same Modbus slave ID, however have differing registers to write to

CASE PumpType OF
	
	E_DosingPump.PH_DOWN:
		getAdrReadWriteSpeed := 16#64;
		
	E_DosingPump.NUTRIENT_A:
		getAdrReadWriteSpeed := 16#65;
		
	E_DosingPump.NUTRIENT_B:
		getAdrReadWriteSpeed := 16#66;
		
	E_DosingPump.NUTRIENT_C:
		getAdrReadWriteSpeed := 16#67;
		
	E_DosingPump.PH_UP:
		getAdrReadWriteSpeed := 16#68;
		
END_CASE
END_METHOD

METHOD init_ModbusRequests : BOOL
VAR_INPUT
END_VAR
stModRead_MotorSpeed.SlaveAddress := nModbusUnitID;			
stModRead_MotorSpeed.AdrFirstSlaveRegisterRead := getAdrReadWriteSpeed(PumpType := ePumpType);
stModRead_MotorSpeed.QtyWordsToRead := 1;				// The value is a 16-bit word
stModRead_MotorSpeed.bRequestAccepted := FALSE;
stModRead_MotorSpeed.bRequestCompleted := FALSE;
stModRead_MotorSpeed.ReadRegsVals := GVL.ModbusEmptyBuffer;

stModRead_MotorRunTime.SlaveAddress := nModbusUnitID;			
stModRead_MotorRunTime.AdrFirstSlaveRegisterRead := getAdrReadAccumRunTime(PumpType := ePumpType);
stModRead_MotorRunTime.QtyWordsToRead := 1;				// The value is a 32-bit word
stModRead_MotorRunTime.bRequestAccepted := FALSE;
stModRead_MotorRunTime.bRequestCompleted := FALSE;
stModRead_MotorRunTime.ReadRegsVals := GVL.ModbusEmptyBuffer;


		
stModWrite_MotorSpeed.SlaveAddress := nModbusUnitID;
stModWrite_MotorSpeed.AdrFirstSlaveRegisterWrite := getAdrReadWriteSpeed(PumpType := ePumpType);
stModWrite_MotorSpeed.bRequestAccepted := FALSE;
stModWrite_MotorSpeed.bRequestCompleted := FALSE;
stModWrite_MotorSpeed.QtyWordsToWrite := 1;

stModWrite_SetID.SlaveAddress := 254;
stModWrite_SetID.AdrFirstSlaveRegisterWrite := 0;
stModWrite_SetID.bRequestAccepted := FALSE;
stModWrite_SetID.bRequestCompleted := FALSE;
stModWrite_SetID.QtyWordsToWrite := 1;
END_METHOD

METHOD readSpeed : BOOL
VAR_INPUT
END_VAR
fbModbusManager.addRequest_Read_Priority(ReadRequest := ADR(stModRead_MotorSpeed));
END_METHOD

METHOD setDoseQTY_InitDose : BOOL
VAR_INPUT
	DoseQtyMls: INT;
END_VAR

nDoseQtyMls := DoseQtyMls;
bInitialDose := TRUE;
END_METHOD

METHOD setModID : BOOL
VAR_INPUT
	DesiredID: UINT;
END_VAR
stModWrite_SetID.WriteRegVals[1] := DesiredID;
fbModbusManager.addRequest_Write_Priority(WriteRequest := ADR(stModWrite_SetID));
END_METHOD

METHOD setOFF : BOOL
VAR_INPUT
	RequestComplete: 	POINTER TO BOOL;
END_VAR
VAR_OUTPUT
	RequestAccepted: 	BOOL;
END_VAR
eSMState := DOSING_OFF_TRIG;
END_METHOD

METHOD setON : BOOL
VAR_INPUT
	RateMlph	 : 		UINT;
	RequestComplete: 	POINTER TO BOOL;
END_VAR

VAR_OUTPUT
	RequestAccepted: 	BOOL;
END_VAR
END_METHOD

METHOD setSpeed99 : BOOL
VAR_INPUT
END_VAR
nPumpSpeed_Requested := 99;
stModWrite_MotorSpeed.WriteRegVals[1] := UINT_TO_WORD(nPumpSpeed_Requested);
fbModbusManager.addRequest_Write_Priority(WriteRequest := ADR(stModWrite_MotorSpeed));
END_METHOD

END_FUNCTION_BLOCK

// ---- POUs/99 Utilities/FB_ModbusManager.TcPOU
FUNCTION_BLOCK FB_ModbusManager

VAR PERSISTENT
	tReadVaisala: 				TIME := T#1.2S;
	tDelay:						TIME := T#75MS;
	tDelayBetweenMsg_Normal:	TIME := T#75MS;
	tDelayBetweenMsg_Slow:		TIME := T#1.2S;	

END_VAR

VAR
	fbModbusMaster: FB_ModbusMaster_R2;
	
	bFirstRun: BOOL := TRUE;
	
	// Regular modbus requests
	aRequests_Read: 			ARRAY[0..(GVL.Max_Modbus_Requests_Read - 1)] OF POINTER TO ST_Modbus_ReadRequest;
	nIterator_Read_Insert: 		INT := 0;
	nIterator_Read_Action: 		INT := 0;
	nTotalRequests_Read: 		INT := 0;
	
	aRequests_Write: 			ARRAY[0..(GVL.Max_Modbus_Requests_Write - 1)] OF POINTER TO ST_Modbus_WriteRequest;
	nIterator_Write_Insert: 	INT := 0;
	nIterator_Write_Action:		INT := 0;
	nTotalRequests_Write: 		INT := 0;
	
	nNumRetries: 				INT := 0;
	bRead_or_Write_0_1:			BOOL := FALSE;
	bRequestAccepted: 			BOOL := FALSE;
	
	eSMState: (WAIT, REQUEST_READ, READING, READ, REQUEST_WRITE, WRITING, WRITTEN, REQUEST_READ_PRIORITY, READING_PRIORITY, READ_PRIORITY, REQUEST_WRITE_PRIORITY, WRITING_PRIORITY, WRITTEN_PRIORITY,REQUEST_READ_2, READING_2, READ_2, ERROR) := WAIT;
	
	fbTON_RequestTimeout: TON := (PT := GVL.ModbusTimeout);

	fbTON_DelayBetweenMSG: TON := (PT := tDelay, IN := FALSE);
	
	
	// These two buffers are for priority messages and will be serviced before requests in the other buffers (similar to QoS)
	aRequests_Read_Priority: 			ARRAY[0..(GVL.Max_Modbus_Requests_Read_Priority - 1)] OF POINTER TO ST_Modbus_ReadRequest;
	nIterator_Read_Insert_Priority: 	INT := 0;
	nIterator_Read_Action_Priority: 	INT := 0;
	nTotalRequests_Read_Priority: 		INT := 0;
	
	aRequests_Write_Priority: 			ARRAY[0..(GVL.Max_Modbus_Requests_Write_Priority - 1)] OF POINTER TO ST_Modbus_WriteRequest;
	nIterator_Write_Insert_Priority: 	INT := 0;
	nIterator_Write_Action_Priority:	INT := 0;
	nTotalRequests_Write_Priority: 		INT := 0;
	
	bRead_or_Write_0_1_Priority:		BOOL := FALSE;
	
	
	
	fbTON_ReadVaisala: TON := (PT := tReadVaisala, IN := FALSE);
	
	// Vaisala Sensor Requests - different modbus card settings
	aRequests_Read_2: 				ARRAY[0..(GVL.Max_Modbus_Requests_Read - 1)] OF POINTER TO ST_Modbus_ReadRequest;
	nIterator_Read_Insert_2: 		INT := 0;
	nIterator_Read_Action_2: 		INT := 0;
	nTotalRequests_Read_2: 			INT := 0;
	
	aRequests_Write_2: 				ARRAY[0..(GVL.Max_Modbus_Requests_Write - 1)] OF POINTER TO ST_Modbus_WriteRequest;
	nIterator_Write_Insert_2: 		INT := 0;
	nIterator_Write_Action_2:		INT := 0;
	nTotalRequests_Write_2: 		INT := 0;
	
	bRead_or_Write_0_1_Priority_2:		BOOL := FALSE;
	
	
END_VAR

fbModbusMaster();
fbTON_RequestTimeout(PT := GVL.ModbusTimeout);

IF bFirstRun THEN
	fbTON_ReadVaisala(IN := TRUE);
	bFirstRun := FALSE;
END_IF


CASE eSMState OF
	
	WAIT:
		// Wait for a message to be received in either the Rx or Tx buffers
		nNumRetries := 0;
		
		fbTON_DelayBetweenMSG(PT := tDelay, IN := TRUE);
		
		IF fbTON_DelayBetweenMSG.Q THEN
			// Service priority writes first
			IF nTotalRequests_Write_Priority > 0 THEN
				eSMState := REQUEST_WRITE_PRIORITY;
			// Service priority reads second
			ELSIF nTotalRequests_Read_Priority > 0 THEN
				eSMState := REQUEST_READ_PRIORITY;
			// Else toggle betwweenm read and write
			ELSIF nTotalRequests_Write > 0 THEN   // If there are no priority messages then serve the non-critical requests
				eSMState := REQUEST_WRITE;
			ELSIF nTotalRequests_Read > 0 THEN
					eSMState := REQUEST_READ;	
			ELSIF nTotalRequests_Read_2 > 0 THEN
					eSMState := REQUEST_READ_2;	
			END_IF
			fbTON_DelayBetweenMSG(IN := FALSE);
		END_IF
		
		bRead_or_Write_0_1 := NOT bRead_or_Write_0_1;

		
	REQUEST_READ:
		fbModbusMaster.readRegs(ReadRequest := aRequests_Read[nIterator_Read_Action], bRequestAccepted => bRequestAccepted);
		IF bRequestAccepted THEN
			eSMState := READING;
			bRequestAccepted := FALSE;
			fbTON_RequestTimeout.IN := TRUE; 
		END_IF
		// Send a read request to the modbus master, progress to READING if modbus master accepts
		
	READING:
	
		IF aRequests_Read[nIterator_Read_Action]^.bRequestCompleted = TRUE THEN
			eSMState := READ;
			fbTON_RequestTimeout.IN := FALSE;
		END_IF
		
		IF fbTON_RequestTimeout.Q THEN
			eSMState := REQUEST_READ; 
			nNumRetries := nNumRetries + 1;
			IF nNumRetries > GVL.ModbusMaxRetires THEN
				// ADD CODE HERE - Raise an error - and proceed to the next request - attach info about the request to the error so we can troubleshoot it
				eSMState := READ;
			END_IF
		END_IF
		
		// Stay in this state until the boolean pointer of job completed is set to true
		// Monitor the timeout timer and retry request if necessary
		
	READ:
		// Set the position in the ring buffer to 0 and iterate to the next, return to wait where the decision will be made to read or write
		aRequests_Read[nIterator_Read_Action] := 0;
		nIterator_Read_Action := nIterator_Read_Action + 1;
		
		IF nIterator_Read_Action > (GVL.Max_Modbus_Requests_Read - 1) THEN // return to 0 index if we are at the end of the buffer
			nIterator_Read_Action := 0;
		END_IF
		nTotalRequests_Read := nTotalRequests_Read - 1;
		eSMState := WAIT;
		tDelay := tDelayBetweenMsg_Normal;
		
	
		
	REQUEST_WRITE:
		// Send a read request to the modbus master, progress to WRITING if modbus master accepts
		fbModbusMaster.writeRegs(WriteRequest := aRequests_Write[nIterator_Write_Action], bRequestAccepted => bRequestAccepted);
		IF bRequestAccepted THEN
			eSMState := WRITING;
			bRequestAccepted := FALSE;
			fbTON_RequestTimeout.IN := TRUE;
		END_IF
		
	WRITING:
		// Stay in this state until the boolean pointer of job completed is set to true
		IF aRequests_Write[nIterator_Write_Action]^.bRequestCompleted = TRUE THEN
			eSMState := WRITTEN;
			fbTON_RequestTimeout.IN := FALSE;
		END_IF
		
		IF fbTON_RequestTimeout.Q THEN
			eSMState := REQUEST_WRITE; 
			nNumRetries := nNumRetries + 1;
			IF nNumRetries > GVL.ModbusMaxRetires THEN
				// ADD CODE HERE - Raise an error - and proceed to the next request - attach info about the request to the error so we can troubleshoot it
				eSMState := WRITTEN;
			END_IF
		END_IF
		
		
	WRITTEN:
		// Set the position in the ring buffer to 0 and iterate to the next, return to wait where the decision will be made to read or write
		aRequests_Write[nIterator_Write_Action] := 0;
		nIterator_Write_Action := nIterator_Write_Action + 1;
		
		IF nIterator_Write_Action > (GVL.Max_Modbus_Requests_Write - 1) THEN
			nIterator_Write_Action := 0;
		END_IF
		
		nTotalRequests_Write := nTotalRequests_Write - 1;
		eSMState := WAIT;
		tDelay := tDelayBetweenMsg_Normal;
		
		
	REQUEST_READ_PRIORITY:
		fbModbusMaster.readRegs(ReadRequest := aRequests_Read_Priority[nIterator_Read_Action_Priority], bRequestAccepted => bRequestAccepted);
		IF bRequestAccepted THEN
			eSMState := READING_PRIORITY;
			bRequestAccepted := FALSE;
			fbTON_RequestTimeout.IN := TRUE;
		END_IF
		// Send a read request to the modbus master, progress to READING if modbus master accepts
		
	READING_PRIORITY:
	
		IF aRequests_Read_Priority[nIterator_Read_Action_Priority]^.bRequestCompleted = TRUE THEN
			eSMState := READ_PRIORITY;
			fbTON_RequestTimeout.IN := FALSE;
		END_IF
		
		IF fbTON_RequestTimeout.Q THEN
			eSMState := REQUEST_READ_PRIORITY; 
			nNumRetries := nNumRetries + 1;
			IF nNumRetries > GVL.ModbusMaxRetires THEN
				// ADD CODE HERE - Raise an error - and proceed to the next request - attach info about the request to the error so we can troubleshoot it
				eSMState := READ_PRIORITY;
			END_IF
		END_IF
		
		// Stay in this state until the boolean pointer of job completed is set to true
		// Monitor the timeout timer and retry request if necessary
		
	READ_PRIORITY:
		// Set the position in the ring buffer to 0 and iterate to the next, return to wait where the decision will be made to read or write
		aRequests_Read_Priority[nIterator_Read_Action_Priority] := 0;
		nIterator_Read_Action_Priority := nIterator_Read_Action_Priority + 1;
		
		IF nIterator_Read_Action_Priority > (GVL.Max_Modbus_Requests_Read_Priority - 1) THEN // return to 0 index if we are at the end of the buffer
			nIterator_Read_Action_Priority := 0;
		END_IF
		nTotalRequests_Read_Priority := nTotalRequests_Read_Priority - 1;
		eSMState := WAIT;
		tDelay := tDelayBetweenMsg_Normal;
	
		
	REQUEST_WRITE_PRIORITY:
		// Send a read request to the modbus master, progress to WRITING if modbus master accepts
		fbModbusMaster.writeRegs(WriteRequest := aRequests_Write_Priority[nIterator_Write_Action_Priority], bRequestAccepted => bRequestAccepted);
		IF bRequestAccepted THEN
			eSMState := WRITING_PRIORITY;
			bRequestAccepted := FALSE;
			fbTON_RequestTimeout.IN := TRUE;
		END_IF
		
	WRITING_PRIORITY:
		// Stay in this state until the boolean pointer of job completed is set to true
		IF aRequests_Write_Priority[nIterator_Write_Action_Priority]^.bRequestCompleted = TRUE THEN
			eSMState := WRITTEN_PRIORITY;
			fbTON_RequestTimeout.IN := FALSE;
		END_IF
		
		IF fbTON_RequestTimeout.Q THEN
			eSMState := REQUEST_WRITE_PRIORITY; 
			nNumRetries := nNumRetries + 1;
			IF nNumRetries > GVL.ModbusMaxRetires THEN
				// ADD CODE HERE - Raise an error - and proceed to the next request - attach info about the request to the error so we can troubleshoot it
				eSMState := WRITTEN_PRIORITY;
			END_IF
		END_IF
		
		
	WRITTEN_PRIORITY:
		// Set the position in the ring buffer to 0 and iterate to the next, return to wait where the decision will be made to read or write
		aRequests_Write_Priority[nIterator_Write_Action_Priority] := 0;
		nIterator_Write_Action_Priority := nIterator_Write_Action_Priority + 1;
		
		IF nIterator_Write_Action_Priority > (GVL.Max_Modbus_Requests_Write_Priority - 1) THEN
			nIterator_Write_Action_Priority := 0;
		END_IF
		
		nTotalRequests_Write_Priority := nTotalRequests_Write_Priority - 1;
		eSMState := WAIT;
		tDelay := tDelayBetweenMsg_Normal;
		
		
	REQUEST_READ_2:
	
	
		// Change the card settings here
		
		fbModbusMaster.readRegs(ReadRequest := aRequests_Read_2[nIterator_Read_Action_2], bRequestAccepted => bRequestAccepted);
		IF bRequestAccepted THEN
			eSMState := READING_2;
			bRequestAccepted := FALSE;
			fbTON_RequestTimeout.IN := TRUE;
		END_IF
		// Send a read request to the modbus master, progress to READING if modbus master accepts
		
	READING_2:
	
		IF aRequests_Read_2[nIterator_Read_Action_2]^.bRequestCompleted = TRUE THEN
			eSMState := READ_2;
			fbTON_RequestTimeout.IN := FALSE;
		END_IF
		
		IF fbTON_RequestTimeout.Q THEN
			eSMState := REQUEST_READ_2; 
			nNumRetries := nNumRetries + 1;
			IF nNumRetries > GVL.ModbusMaxRetires THEN
				// ADD CODE HERE - Raise an error - and proceed to the next request - attach info about the request to the error so we can troubleshoot it
				eSMState := READ_2;
			END_IF
		END_IF
		
		// Stay in this state until the boolean pointer of job completed is set to true
		// Monitor the timeout timer and retry request if necessary
		
	READ_2:
		// Set the position in the ring buffer to 0 and iterate to the next, return to wait where the decision will be made to read or write
		aRequests_Read_2[nIterator_Read_Action_2] := 0;
		nIterator_Read_Action_2 := nIterator_Read_Action_2 + 1;
		
		IF nIterator_Read_Action_2 > (GVL.Max_Modbus_Requests_Read - 1) THEN // return to 0 index if we are at the end of the buffer
			nIterator_Read_Action_2 := 0;
		END_IF
		nTotalRequests_Read_2 := nTotalRequests_Read_2 - 1;
		

		eSMState := WAIT;
				// Set the position in the ring buffer to 0 and iterate to the next, return to wait where the decision will be made to read or write
		tDelay := tDelayBetweenMsg_Slow;

		
	ERROR:
		//
		
END_CASE

METHOD addRequest_Read : BOOL
VAR_INPUT
	ReadRequest: POINTER TO ST_Modbus_ReadRequest;
END_VAR
IF aRequests_Read[nIterator_Read_Insert] = 0 THEN
	
	aRequests_Read[nIterator_Read_Insert] := ReadRequest;
	aRequests_Read[nIterator_Read_Insert]^.bRequestAccepted := FALSE;
	aRequests_Read[nIterator_Read_Insert]^.bRequestCompleted := FALSE;
	nIterator_Read_Insert := nIterator_Read_Insert + 1;
	
	IF nIterator_Read_Insert > (GVL.Max_Modbus_Requests_Read -1) THEN
		nIterator_Read_Insert := 0;
	END_IF
	
	nTotalRequests_Read := nTotalRequests_Read + 1;
	
	
	addRequest_Read := TRUE;
ELSE
	addRequest_Read := FALSE;	// A buffer overflow has occured here, add some error raising code here
END_IF
END_METHOD

METHOD addRequest_Read_Priority : BOOL
VAR_INPUT
	ReadRequest: POINTER TO ST_Modbus_ReadRequest;
END_VAR
IF aRequests_Read_Priority[nIterator_Read_Insert_Priority] = 0 THEN
	
	aRequests_Read_Priority[nIterator_Read_Insert_Priority] := ReadRequest;
	aRequests_Read_Priority[nIterator_Read_Insert_Priority]^.bRequestAccepted := FALSE;
	aRequests_Read_Priority[nIterator_Read_Insert_Priority]^.bRequestCompleted := FALSE;
	nIterator_Read_Insert_Priority := nIterator_Read_Insert_Priority + 1;
	
	IF nIterator_Read_Insert_Priority > (GVL.Max_Modbus_Requests_Read_Priority -1) THEN
		nIterator_Read_Insert_Priority := 0;
	END_IF
	
	nTotalRequests_Read_Priority := nTotalRequests_Read_Priority + 1;
	
	
	addRequest_Read_Priority := TRUE;
ELSE
	addRequest_Read_Priority := FALSE;	// A buffer overflow has occured here, add some error raising code here
END_IF
END_METHOD

METHOD addRequest_Read_Vaisala : BOOL
VAR_INPUT
	ReadRequest: POINTER TO ST_Modbus_ReadRequest;
END_VAR
IF aRequests_Read_2[nIterator_Read_Insert_2] = 0 THEN
	
	aRequests_Read_2[nIterator_Read_Insert_2] := ReadRequest;
	aRequests_Read_2[nIterator_Read_Insert_2]^.bRequestAccepted := FALSE;
	aRequests_Read_2[nIterator_Read_Insert_2]^.bRequestCompleted := FALSE;
	nIterator_Read_Insert_2 := nIterator_Read_Insert_2 + 1;
	
	IF nIterator_Read_Insert_2 > (GVL.Max_Modbus_Requests_Read -1) THEN
		nIterator_Read_Insert_2 := 0;
	END_IF
	
	nTotalRequests_Read_2 := nTotalRequests_Read_2 + 1;
	
	
	addRequest_Read_Vaisala := TRUE;
ELSE
	addRequest_Read_Vaisala := FALSE;	// A buffer overflow has occured here, add some error raising code here
END_IF
END_METHOD

METHOD addRequest_Write : BOOL
VAR_INPUT
	WriteRequest: POINTER TO ST_Modbus_WriteRequest;
END_VAR
IF aRequests_Write[nIterator_Write_Action] = 0 THEN
	aRequests_Write[nIterator_Write_Action] := WriteRequest;
	aRequests_Write[nIterator_Write_Action]^.bRequestAccepted := FALSE;
	aRequests_Write[nIterator_Write_Action]^.bRequestCompleted := FALSE;
	nIterator_Write_Insert := nIterator_Write_Insert + 1;
	
	IF nIterator_Write_Insert > (GVL.Max_Modbus_Requests_Write - 1) THEN
		nIterator_Write_Insert := 0;
	END_IF
	
	nTotalRequests_Write := nTotalRequests_Write + 1;
	
ELSE
	addRequest_Write := FALSE; // A buffer overflow has occured here, add some error raising code here
END_IF
END_METHOD

METHOD addRequest_Write_Priority : BOOL
VAR_INPUT
	WriteRequest: POINTER TO ST_Modbus_WriteRequest;
END_VAR
IF aRequests_Write_Priority[nIterator_Write_Insert_Priority] = 0 THEN
	
	aRequests_Write_Priority[nIterator_Write_Insert_Priority] := WriteRequest;
	aRequests_Write_Priority[nIterator_Write_Insert_Priority]^.bRequestAccepted := FALSE;
	aRequests_Write_Priority[nIterator_Write_Insert_Priority]^.bRequestCompleted := FALSE;
	nIterator_Write_Insert_Priority := nIterator_Write_Insert_Priority + 1;
	
	IF nIterator_Write_Insert_Priority > (GVL.Max_Modbus_Requests_Write_Priority - 1) THEN
		nIterator_Write_Insert_Priority := 0;
	END_IF
	
	nTotalRequests_Write_Priority := nTotalRequests_Write_Priority + 1;
	
ELSE
	addRequest_Write_Priority := FALSE; // A buffer overflow has occured here, add some error raising code here
END_IF
END_METHOD

METHOD FB_init : BOOL
VAR_INPUT
	bInitRetains : BOOL; // if TRUE, the retain variables are initialized (warm start / cold start)
	bInCopyCode : BOOL;  // if TRUE, the instance afterwards gets moved into the copy code (online change)
END_VAR

VAR
	i: INT := 0;
END_VAR
WHILE i < GVL.Max_Modbus_Requests_Read DO
	aRequests_Read[i] := 0;
	i := i + 1;
END_WHILE

i := 0;

WHILE i < GVL.Max_Modbus_Requests_Write DO
	aRequests_Write[i] := 0;
	i := i + 1;
END_WHILE
END_METHOD

END_FUNCTION_BLOCK

// ---- POUs/99 Utilities/FB_ModbusMaster_R2.TcPOU
FUNCTION_BLOCK FB_ModbusMaster_R2

VAR
	bFirstRun: BOOL := TRUE;
	
	MB: ModbusRtuMaster_KL6x22B;
	
	nReadRegsVals: POINTER TO ARRAY[1..10] OF WORD;
	nWriteRegVals: ARRAY[1..10] OF WORD;
	
	bRequestFinshed : POINTER TO BOOL;
		
	nSlaveAddress : BYTE;
	nQtyWordsToRead : WORD;
	nQtyWordsToWrite : WORD;
	nAdrFirstSlaveRegisterRead : WORD;
	nAdrFirstSlaveRegisterWrite : WORD;
	nTimeout : TIME := T#1S;
	
	// State Machine
	eState: (RESET, WAIT, READ_TRIG, READ, WRITE_TRIG, WRITE) := WAIT;
	bBusy: BOOL;
	
	//eOperationType: (READ_OP, WRITE_OP, READWRITE_OP);
	eOperationType: E_AccessType;
	fbTrigger : R_TRIG;
	
		
	
END_VAR

fbTrigger();
MB();







CASE eState OF
	

	WAIT :
		MB.ReadRegs(Execute := FALSE);
        MB.WriteRegs(Execute := FALSE);
		
		IF fbTrigger.Q THEN
			IF eOperationType = E_AccessType.WRITE THEN
				eState := WRITE_TRIG;
			ELSIF eOperationType = E_AccessType.READ THEN
				eState := READ_TRIG;
			END_IF
		END_IF
		
		
		
		
	READ_TRIG : 
		
		 MB.ReadRegs(
			UnitID:= nSlaveAddress, 
			Quantity:= nQtyWordsToRead, 
			MBAddr:= nAdrFirstSlaveRegisterRead, 
			cbLength:= nQtyWordsToRead * 2,//SIZEOF(nReadRegsVals), 
			pMemoryAddr:= ADR(nReadRegsVals^), 
			Execute:= TRUE, 
			Timeout:= nTimeout );
		
		
		IF NOT MB.BUSY THEN 
			MB.ReadRegs(Execute := FALSE );
			bBusy := TRUE;
			IF MB.Error THEN 
				eState := READ;           // handle errors 
			ELSE 
				eState := READ; // [...]               // keep going 
			END_IF
		END_IF

		
		
	READ :
	
		IF NOT MB.BUSY OR MB.Error THEN
			eState := WAIT;
			bRequestFinshed^ := TRUE;
			bBusy := FALSE;
			fbTrigger.CLK := FALSE;
			
		END_IF
	

		
	WRITE_TRIG :
			
		MB.UnitID:= nSlaveAddress;
		MB.Quantity:=1;
		MB.MBAddr:= nAdrFirstSlaveRegisterWrite;
		MB.cbLength:= nQtyWordsToWrite * 2;
		MB.pMemoryAddr:= ADR(nWriteRegVals);
		MB.Execute:= TRUE;
		MB.Timeout:= nTimeout;
		MB.WriteSingleRegister();

			
		IF NOT MB.BUSY THEN 
			//MB.WriteRegs(Execute := FALSE );
			MB.Execute := FALSE;
			bBusy := TRUE;
			IF MB.Error THEN 
				eState := WRITE;           				// handle errors 
			ELSE 
				eState := WRITE;			            // keep going 
			END_IF
		END_IF

	
	WRITE :
		IF NOT MB.BUSY OR MB.Error THEN
			eState := WAIT;
			bRequestFinshed^ := TRUE;
			bBusy := FALSE;
			fbTrigger.CLK := FALSE;
			
		END_IF

END_CASE

METHOD Error : BOOL
VAR_INPUT
END_VAR
Error := MB.Error;
END_METHOD

METHOD FB_init : BOOL
VAR_INPUT
	bInitRetains : BOOL; // if TRUE, the retain variables are initialized (warm start / cold start)
	bInCopyCode : BOOL;  // if TRUE, the instance afterwards gets moved into the copy code (online change)
END_VAR
END_METHOD

METHOD isBusy : BOOL
isBusy := bBusy;
END_METHOD

METHOD readRegs : BOOL
VAR_INPUT
	ReadRequest: POINTER TO ST_Modbus_ReadRequest;
END_VAR

VAR_OUTPUT
	bRequestAccepted: BOOL;
END_VAR
IF eState = WAIT THEN
	eOperationType := E_AccessType.READ;
	nReadRegsVals := ADR(ReadRequest^.ReadRegsVals);
	nSlaveAddress := UINT_TO_BYTE(ReadRequest^.SlaveAddress);
	nQtyWordsToRead := UINT_TO_WORD(ReadRequest^.QtyWordsToRead);
	nAdrFirstSlaveRegisterRead := UINT_TO_WORD(ReadRequest^.AdrFirstSlaveRegisterRead);
	fbTrigger.CLK := TRUE;
	bRequestAccepted := TRUE;
	bBusy := TRUE;
	bRequestFinshed := ADR(ReadRequest^.bRequestCompleted);
END_IF
END_METHOD

METHOD writeReg : BOOL
VAR_INPUT
	WriteRegVal: WORD;
	SlaveAddress : UINT;
	AdrFirstSlaveRegisterWrite : UINT;
	bRequestCompleted : POINTER TO BOOL;
	
	WriteRequest: ST_Modbus_WriteRequest;
END_VAR

VAR_OUTPUT
	bRequestAccepted: BOOL := FALSE;
END_VAR
(* IF eState = WAIT THEN
	eOperationType := E_AccessType.WRITE;
	//nWriteRegVals[0] := WriteRegVal;
	nWriteRegVals[1] := WriteRegVal;
	nWriteRegVals[1] := WriteRequest.
	nSlaveAddress := UINT_TO_BYTE(SlaveAddress);
	nQtyWordsToWrite := 1;
	nAdrFirstSlaveRegisterWrite := UINT_TO_BYTE(AdrFirstSlaveRegisterWrite);
	bRequestAccepted := TRUE;
	bRequestFinshed := bRequestCompleted;
	fbTrigger.CLK := TRUE;
	eState := WRITE_TRIG;
	
END_IF
*) 

// This needs to be re written to suit ST requests
END_METHOD

METHOD writeRegs : BOOL
VAR_INPUT

	
	WriteRequest: POINTER TO ST_Modbus_WriteRequest;

END_VAR

VAR_OUTPUT
	bRequestAccepted: BOOL := FALSE;
END_VAR
IF eState = WAIT THEN
	eOperationType := E_AccessType.WRITE;
	nWriteRegVals := WriteRequest^.WriteRegVals;
	nSlaveAddress := UINT_TO_BYTE(WriteRequest^.SlaveAddress);
	nQtyWordsToWrite := UINT_TO_WORD(WriteRequest^.QtyWordsToWrite);
	nAdrFirstSlaveRegisterWrite := UINT_TO_WORD(WriteRequest^.AdrFirstSlaveRegisterWrite);
	bRequestFinshed := ADR(WriteRequest^.bRequestCompleted);	
	fbTrigger.CLK := TRUE;
	bRequestAccepted := TRUE;
	
	eState := WRITE_TRIG;
END_IF
END_METHOD

END_FUNCTION_BLOCK

// ---- POUs/01 Actuators/Dosing Machine/FB_DosingPumpAgrowtek_R2_1.TcPOU
{attribute 'OPC.UA.DA.StructuredType' := '1'}
FUNCTION_BLOCK FB_DosingPumpAgrowtek_R2_1 EXTENDS FB_BaseDevice IMPLEMENTS I_PumpDosing

VAR_IN_OUT
	{attribute 'OPC.UA.DA' := '0'}
	//fbModbusMaster: FB_ModbusMaster;
	fbModbusManager: FB_ModbusManager;
END_VAR

VAR_INPUT
	nModbusUnitID: UINT; 
END_VAR

VAR
	// Modbus Variables
	nPumpID: UINT;	// Pump ID is different to the modbus ID because there are 5 pumps on the 1 modbus address
	 
	ePumpType: E_DosingPump;

	
	bEnableComms: BOOL := TRUE;
	bFirtRun: BOOL := TRUE;
	bResetTimer: BOOL := TRUE;
	
	// Async Statemachine Variables
	{attribute 'OPC.UA.DA' := '0'}
	eSMState: (WAIT, DOSING_TRIG, DOSING, DOSING_OFF_TRIG, DOSED);
	
	// Dosing Variables
	{attribute 'OPC.UA.DA' := '0'} 
	fbTONdoseTime: TON;  
	{attribute 'OPC.UA.DA' := '1'} 
	nDoseRateMLph: UINT;
	{attribute 'OPC.UA.DA' := '1'} 
	nDoseQtyMls: REAL;
	{attribute 'OPC.UA.DA' := '1'} 
	tTimeToDose: TIME;
	
	// delay between writing pump speed and reading pump speed
	fbTONreadDelay : TON := (PT := T#1S);

	// Variables updated over Modbus
	{attribute 'OPC.UA.DA' := '1'} 
	nPumpSpeed_Requested: UINT;
	
	{attribute 'OPC.UA.DA' := '1'} 
	nPumpSpeed: UINT;
	{attribute 'OPC.UA.DA' := '1'} 
	nPumpRunTime: UINT; 
	
	tDataRefresh: TIME := T#10S;
	fbTON_DataRefresh: 	TON := (PT := tDataRefresh, IN := FALSE);
	fbTON_MsgTimeout: 	TON := (PT := T#4S, IN := FALSE);
	
	// Modbus Requests
	stModRead_MotorSpeed: 	ST_Modbus_ReadRequest;
	stModRead_MotorRunTime: ST_Modbus_ReadRequest;
	stModWrite_MotorSpeed: 	ST_Modbus_WriteRequest;
	stModWrite_SetID: 		ST_Modbus_WriteRequest;
	
	
	bRaiseError1: BOOL := FALSE;
	bClearError: BOOL := FALSE;
	bRaiseError2: BOOL := FALSE;
	
	
END_VAR

fbTONdoseTime();
fbTON_MsgTimeout();
fbTON_DataRefresh();
fbTONreadDelay();

IF GVL.bAutoUpdateDeviceState THEN
	eState := eStateTarget;	
END_IF

IF bFirtRun THEN
	init_ModbusRequests();
	bFirtRun := FALSE;
END_IF

IF eMode = E_DeviceMode.MANUAL THEN
	bEnable := TRUE;
END_IF
(*

IF bEnable AND eStateTarget = E_DeviceState.ON AND eState <> E_DeviceState.RUNNING THEN
		eSMState := WAIT;
END_IF

IF (bEnable = FALSE OR eStateTarget = E_DeviceState.IDLE) AND eState <> E_DeviceState.IDLE THEN
		eSMState := 0;
END_IF
*)


IF bResetTimer THEN
	fbTON_DataRefresh.IN := TRUE;
	bResetTimer := FALSE;
END_IF

// Asynchronous update of local variables from the Modbus request structures
nPumpSpeed 		:= WORD_TO_UINT(stModRead_MotorSpeed.ReadRegsVals[1]);
nPumpRunTime 	:= WORD_TO_UINT(stModRead_MotorRunTime.ReadRegsVals[1]);
	
// Request update of local veriables every Xs (in accordance with adjustable DataRefresh timer)
(*IF fbTON_DataRefresh.Q AND bEnable THEN // AND bEnableComms THEN
	// fbModbusManager.addRequest_Read_Priority(ReadRequest := ADR(stModRead_MotorRunTime));
	fbModbusManager.addRequest_Read_Priority(ReadRequest := ADR(stModRead_MotorSpeed));
	fbTON_DataRefresh.IN := FALSE;
	bResetTimer := TRUE;
END_IF
*)


// Statemachine to handle dosing commands
//IF eState = E_Devicestate.RUNNING THEN //AND bEnableComms THEN
	CASE eSMState OF
	
		WAIT:
			// Wait for a dosing command
			eState := E_DeviceState.IDLE;
			// Beau make sure the timeout timer is cleared in case it was left on last time
			fbTON_MsgTimeout.IN := FALSE;
			
		DOSING_TRIG:
			// A call to the 'executeDose' has been received, send modbus command
			// Send the dosing modbus request and start the timer
			//nPumpSpeed_Requested := 100;
			stModWrite_MotorSpeed.WriteRegVals[1] := UINT_TO_WORD(nPumpSpeed_Requested);
			fbModbusManager.addRequest_Write_Priority(WriteRequest := ADR(stModWrite_MotorSpeed));
			// Beau instead of reading pump speed immediately, start the delay timer
			fbTONreadDelay.IN := TRUE;
			//fbModbusManager.addRequest_Read_Priority(ReadRequest := ADR(stModRead_MotorSpeed));
			fbTONdoseTime.IN := TRUE;
			fbTON_MsgTimeout.PT := fbTONdoseTime.PT + T#1S;
			fbTON_MsgTimeout.IN := TRUE;
			eSMState := DOSING;
			eState := E_DeviceState.RUNNING;
			
	
		DOSING: 
		
			// Beau try to read pump speed one second after writing pump speed
			IF fbTONreadDelay.Q THEN
				fbModbusManager.addRequest_Read_Priority(ReadRequest := ADR(stModRead_MotorSpeed));	
				// reset the timer so we don't send another read request
				fbTONreadDelay.IN := FALSE;
			END_IF
			
			IF fbTON_MsgTimeout.Q AND NOT (nPumpSpeed_Requested = nPumpSpeed) THEN
				// The pump hasn't turned on after it was requested to - try again!
				fbModbusManager.addRequest_Read_Priority(ReadRequest := ADR(stModRead_MotorSpeed));
				fbTONdoseTime.IN := FALSE;
				fbTON_MsgTimeout.IN := FALSE;
				eSMState := DOSING_TRIG; // go back and retry
			END_IF
			
			
			IF fbTONdoseTime.Q THEN
				fbTONdoseTime.IN := FALSE; // reset the timer
				IF nPumpSpeed = nPumpSpeed_Requested THEN
					fbTONdoseTime.IN := FALSE;
					fbTON_MsgTimeout.IN := FALSE;
					eSMState := DOSING_OFF_TRIG; // the pump turned on, now we can turn off
				END_IF
			END_IF
			eState := E_DeviceState.RUNNING;
				
			
		DOSING_OFF_TRIG:
			
			// Monitor the run time / compare against the calculated dosing time
			// when dosing time has been exceeded move to dosed
			nPumpSpeed_Requested := 0; // turn the pump off
			stModWrite_MotorSpeed.WriteRegVals[1] := UINT_TO_WORD(nPumpSpeed_Requested);
			
			fbModbusManager.addRequest_Write_Priority(WriteRequest := ADR(stModWrite_MotorSpeed));
			
			fbModbusManager.addRequest_Read_Priority(ReadRequest := ADR(stModRead_MotorSpeed));
			
			fbModbusManager.addRequest_Write_Priority(WriteRequest := ADR(stModWrite_MotorSpeed));
			fbModbusManager.addRequest_Write_Priority(WriteRequest := ADR(stModWrite_MotorSpeed));
			fbModbusManager.addRequest_Write_Priority(WriteRequest := ADR(stModWrite_MotorSpeed));
			fbTON_MsgTimeout.IN := TRUE;
			fbTON_MsgTimeout.PT := T#1s;;
			eSMState := DOSED;
			eState := E_DeviceState.RUNNING;
			
			
		DOSED: 
			// Confirm that the pump has stopped by reading the pump speed 
			// go back to wait if the pump speed has reached 0
			
			IF fbTON_MsgTimeout.Q THEN
				fbTON_MsgTimeout.IN := FALSE;
				IF NOT(nPumpSpeed_Requested = nPumpSpeed) THEN
					// The pump hasn't turned off after it was requested to - try again!
					eSMState := DOSING_OFF_TRIG; // go back and retry
				ELSIF nPumpSpeed_Requested = nPumpSpeed THEN
					eSMState := WAIT; // go back to waiting for the next dose
					nDoseQtyMls := 0; // reset this to 0 for SCADA 
				END_IF
			END_IF
			
			// eSMState := WAIT;
			
	
	END_CASE

//END_IF

{warning 'add method implementation '}
METHOD executeDose : BOOL
VAR_INPUT
	DoseQtyMls: LREAL;
	DoseRateMlph: UINT;
	RequestComplete: 	POINTER TO BOOL;
END_VAR
VAR_OUTPUT
	RequestAccepted: BOOL;
END_VAR
(* setDose dispenses the amount requested at a user requested dose rate *)

//nDoseQtyMls := REAL_TO_UINT((UINT_TO_REAL(DoseQtyMls)/10000.0));
IF (bEnable AND bEnableComms) OR (eMode = E_DeviceMode.MANUAL)  THEN
	// nDoseQtyMls := ABS(DoseQtyMls);

	// IF nDoseQtyMls > 1.0 THEN
	
		nPumpSpeed_Requested := 40;
		//tTimeToDose := REAL_TO_TIME(( nDoseQtyMls / (480.0*(UINT_TO_REAL(nPumpSpeed_Requested)/100.0))) * 60.0 *1000.0);  // Agrowtek maximum flow rate is 480 ml/min
		tTimeToDose := REAL_TO_TIME(( ABS(DoseQtyMls) / (480.0*(UINT_TO_REAL(nPumpSpeed_Requested)/100.0))) * 60.0 *1000.0);  // Agrowtek maximum flow rate is 480 ml/min
		//tTimeToDose := REAL_TO_TIME((((UINT_TO_REAL(nDoseQtyMls)) / 480) * 60.0)*1000);  // Agrowtek maximum flow rate is 480 ml/min
		fbTONdoseTime.PT := tTimeToDose;
	
		IF tTimeToDose >= T#1S THEN
			nDoseQtyMls := ABS(DoseQtyMls);
			eSMState 	:= DOSING_TRIG;
			eState 		:= E_Devicestate.RUNNING;
			bBusy 		:= TRUE;	
		END_IF
	END_IF
END_METHOD

METHOD FB_init : BOOL


VAR_INPUT
	bInitRetains : BOOL; // if TRUE, the retain variables are initialized (warm start / cold start)
	bInCopyCode : BOOL;  // if TRUE, the instance afterwards gets moved into the copy code (online change)
	
	PumpID: STRING;
	PumpDescription: STRING;
	PumpType: E_DosingPump;
	ManifoldModbusID: UINT; 
	
END_VAR
sID := PumpID;
sDescr := PumpDescription;
ePumpType := PumpType;
nModbusUnitID := ManifoldModbusID;
END_METHOD

METHOD getAdrReadAccumRunTime : UINT
VAR_INPUT
	PumpType: E_DosingPump;
END_VAR

VAR
	Address: UINT;
END_VAR
// This method retrieves the Modbus register for the individual Agrowtek pump
// We need to do this because 5 pumps share the same Modbus slave ID, however have differing registers to write to

CASE PumpType OF
	
	E_DosingPump.PH_DOWN:
		Address := 16#64;
		
	E_DosingPump.NUTRIENT_A:
		Address := 16#65;
		
	E_DosingPump.NUTRIENT_B:
		Address := 16#66;

	E_DosingPump.NUTRIENT_C:
		Address := 16#67;
		
	E_DosingPump.PH_UP:
		Address := 16#68;
		
END_CASE

getAdrReadAccumRunTime := Address;
END_METHOD

METHOD getAdrReadWriteSpeed : UINT
VAR_INPUT
	PumpType: E_DosingPump;
END_VAR
// This method retrieves the Modbus register for the individual Agrowtek pump
// We need to do this because 5 pumps share the same Modbus slave ID, however have differing registers to write to

CASE PumpType OF
	
	E_DosingPump.PH_DOWN:
		getAdrReadWriteSpeed := 16#64;
		
	E_DosingPump.NUTRIENT_A:
		getAdrReadWriteSpeed := 16#65;
		
	E_DosingPump.NUTRIENT_B:
		getAdrReadWriteSpeed := 16#66;
		
	E_DosingPump.NUTRIENT_C:
		getAdrReadWriteSpeed := 16#67;
		
	E_DosingPump.PH_UP:
		getAdrReadWriteSpeed := 16#68;
		
END_CASE
END_METHOD

METHOD init_ModbusRequests : BOOL
VAR_INPUT
END_VAR
stModRead_MotorSpeed.SlaveAddress := nModbusUnitID;			
stModRead_MotorSpeed.AdrFirstSlaveRegisterRead := getAdrReadWriteSpeed(PumpType := ePumpType);
stModRead_MotorSpeed.QtyWordsToRead := 1;				// The value is a 16-bit word
stModRead_MotorSpeed.bRequestAccepted := FALSE;
stModRead_MotorSpeed.bRequestCompleted := FALSE;
stModRead_MotorSpeed.ReadRegsVals := GVL.ModbusEmptyBuffer;

stModRead_MotorRunTime.SlaveAddress := nModbusUnitID;			
stModRead_MotorRunTime.AdrFirstSlaveRegisterRead := getAdrReadAccumRunTime(PumpType := ePumpType);
stModRead_MotorRunTime.QtyWordsToRead := 1;				// The value is a 32-bit word
stModRead_MotorRunTime.bRequestAccepted := FALSE;
stModRead_MotorRunTime.bRequestCompleted := FALSE;
stModRead_MotorRunTime.ReadRegsVals := GVL.ModbusEmptyBuffer;


		
stModWrite_MotorSpeed.SlaveAddress := nModbusUnitID;
stModWrite_MotorSpeed.AdrFirstSlaveRegisterWrite := getAdrReadWriteSpeed(PumpType := ePumpType);
stModWrite_MotorSpeed.bRequestAccepted := FALSE;
stModWrite_MotorSpeed.bRequestCompleted := FALSE;
stModWrite_MotorSpeed.QtyWordsToWrite := 1;

stModWrite_SetID.SlaveAddress := 254;
stModWrite_SetID.AdrFirstSlaveRegisterWrite := 0;
stModWrite_SetID.bRequestAccepted := FALSE;
stModWrite_SetID.bRequestCompleted := FALSE;
stModWrite_SetID.QtyWordsToWrite := 1;
END_METHOD

METHOD readSpeed : BOOL
VAR_INPUT
END_VAR
fbModbusManager.addRequest_Read_Priority(ReadRequest := ADR(stModRead_MotorSpeed));
END_METHOD

METHOD setModID : BOOL
VAR_INPUT
	DesiredID: UINT;
END_VAR
stModWrite_SetID.WriteRegVals[1] := DesiredID;
fbModbusManager.addRequest_Write_Priority(WriteRequest := ADR(stModWrite_SetID));
END_METHOD

METHOD setOFF : BOOL
VAR_INPUT
	RequestComplete: 	POINTER TO BOOL;
END_VAR
VAR_OUTPUT
	RequestAccepted: 	BOOL;
END_VAR
eSMState := DOSING_OFF_TRIG;
END_METHOD

METHOD setON : BOOL
VAR_INPUT
	RateMlph	 : 		UINT;
	RequestComplete: 	POINTER TO BOOL;
END_VAR

VAR_OUTPUT
	RequestAccepted: 	BOOL;
END_VAR
END_METHOD

METHOD setSpeed99 : BOOL
VAR_INPUT
END_VAR
nPumpSpeed_Requested := 99;
stModWrite_MotorSpeed.WriteRegVals[1] := UINT_TO_WORD(nPumpSpeed_Requested);
fbModbusManager.addRequest_Write_Priority(WriteRequest := ADR(stModWrite_MotorSpeed));
END_METHOD

END_FUNCTION_BLOCK

// ---- POUs/01 Actuators/Dosing Machine/FB_DosingPumpAgrowtek_R2_Batch.TcPOU
{attribute 'OPC.UA.DA.StructuredType' := '1'}
FUNCTION_BLOCK FB_DosingPumpAgrowtek_R2_Batch EXTENDS FB_BaseDevice IMPLEMENTS I_PumpDosing

VAR_IN_OUT
	{attribute 'OPC.UA.DA' := '0'}
	//fbModbusMaster: FB_ModbusMaster;
	fbModbusManager: FB_ModbusManager;
	
	bInitialDose: BOOL := FALSE; // this is set to TRUE when the nDoseQTYMls is pre-loaded for the initial dose sequence. Setting nDoseQtyML or executing doses from control loops is disabled when this is true
END_VAR

VAR_INPUT
	nModbusUnitID: UINT; 
END_VAR

VAR
	// Modbus Variables
	nPumpID: UINT;	// Pump ID is different to the modbus ID because there are 5 pumps on the 1 modbus address
	 
	ePumpType: E_DosingPump;

	
	bEnableComms: BOOL := TRUE;
	bFirtRun: BOOL := TRUE;
	bResetTimer: BOOL := TRUE;
	
	// Async Statemachine Variables
	{attribute 'OPC.UA.DA' := '0'}
	eSMState: (WAIT, SET_TIME, GET_TIME, SET_SPEED, FINISH);
	
	// Dosing Variables
	{attribute 'OPC.UA.DA' := '0'} 
	fbTONdoseTime: TON;  
	{attribute 'OPC.UA.DA' := '1'} 
	nDoseRateMLph: UINT;
	{attribute 'OPC.UA.DA' := '1'} 
	nDoseQtyMls: REAL;
	{attribute 'OPC.UA.DA' := '1'} 
	tTimeToDose: TIME;
	
	nTimeToDoseSeconds: INT;
	nRetries: INT := 0;
	
	// delay between writing pump speed and reading pump speed
	fbTON_WaitForMsg : TON := (PT := T#1S);

	// Variables updated over Modbus
	{attribute 'OPC.UA.DA' := '1'} 
	nPumpSpeed_Requested: UINT;
	
	{attribute 'OPC.UA.DA' := '1'} 
	nPumpSpeed: UINT;
	{attribute 'OPC.UA.DA' := '1'} 
	nPumpRunTime: UINT; 
	
	
	
	
	bDoseRequestSent:		BOOL := FALSE;
	bDoseRequestComplete: 	BOOL := FALSE;
	
	tDataRefresh: TIME := T#10S;
	fbTON_DataRefresh: 	TON := (PT := tDataRefresh, IN := FALSE);
	fbTON_MsgTimeout: 	TON := (PT := T#4S, IN := FALSE);
	
	// Modbus Requests
	stModRead_MotorSpeed: 	ST_Modbus_ReadRequest;
	stModRead_MotorRunTime: ST_Modbus_ReadRequest;
	stModWrite_MotorSpeed: 	ST_Modbus_WriteRequest;
	stModWrite_SetID: 		ST_Modbus_WriteRequest;
	stModWrite_Timeout:	ST_Modbus_WriteRequest;
	stModRead_Timeout:	ST_Modbus_ReadRequest;
	
	
	bRaiseError1: BOOL := FALSE;
	bClearError: BOOL := FALSE;
	bRaiseError2: BOOL := FALSE;
	
	
END_VAR

fbTONdoseTime();
fbTON_MsgTimeout();
fbTON_DataRefresh();
fbTON_WaitForMsg();

IF GVL.bAutoUpdateDeviceState THEN
	eState := eStateTarget;	
END_IF

IF (eStateTarget = E_DeviceState.RUNNING) AND (eState := E_DeviceState.IDLE) THEN  // this is used to handle the initial batch dose commands from the sequene manager (this control loop uses the executeDOse method
	executeDose(DoseQtyMls := nDoseQtyMls, DoseRateMlph := 40, RequestComplete := ADR(bDoseRequestSent));
	eState := E_DeviceState.RUNNING;
END_IF


IF bFirtRun THEN
	init_ModbusRequests();
	bFirtRun := FALSE;
END_IF

IF eMode = E_DeviceMode.MANUAL THEN
	bEnable := TRUE;
END_IF


IF bResetTimer THEN
	fbTON_DataRefresh.IN := TRUE;
	bResetTimer := FALSE;
END_IF

// Asynchronous update of local variables from the Modbus request structures
nPumpSpeed 		:= WORD_TO_UINT(stModRead_MotorSpeed.ReadRegsVals[1]);
nPumpRunTime 	:= WORD_TO_UINT(stModRead_MotorRunTime.ReadRegsVals[1]);
	

CASE eSMState OF

	WAIT:
		eState := E_DeviceState.IDLE;
		fbTON_WaitForMsg(IN := FALSE);
		
	SET_TIME:
		eState := E_DeviceState.RUNNING;
		stModWrite_Timeout.WriteRegVals[1] := INT_TO_WORD(nTimeToDoseSeconds);
		fbModbusManager.addRequest_Write_Priority(WriteRequest := ADR(stModWrite_Timeout));
		fbTON_WaitForMsg(IN := TRUE);
		eSMState := GET_TIME;
		
		
	GET_TIME:
		IF stModRead_Timeout.ReadRegsVals[1] = INT_TO_WORD(nTimeToDoseSeconds) THEN
			stModRead_Timeout.ReadRegsVals[1] := 0;
			fbTON_WaitForMsg(IN := FALSE);
			eSMState := SET_SPEED;
		ELSE
			fbTON_WaitForMsg(IN := TRUE);
		END_IF
	
		IF fbTON_WaitForMsg.Q THEN
			fbModbusManager.addRequest_Read_Priority(ReadRequest := ADR(stModRead_Timeout));	
			fbTON_WaitForMsg(IN := FALSE);
		ELSE
			fbTON_WaitForMsg(IN := FALSE);			// add retry counter here
			nRetries := nRetries + 1;
			IF nRetries > 5 THEN
				eSMState := WAIT;
				eState := E_DeviceState.IDLE;
				bBusy := FALSE;
				nRetries := 0;
				raiseAlarm(Priority := E_AlarmPriority.High, Label := 'Motor Failed to Receive Duration Command After 5 Retries', Enabled := TRUE, DeviceAlarmID := 1);
			END_IF
		END_IF
		
	SET_SPEED:
		fbTON_WaitForMsg(IN := TRUE);
		
		IF fbTON_WaitForMsg.Q THEN
			stModWrite_MotorSpeed.WriteRegVals[1] := UINT_TO_WORD(nPumpSpeed_Requested);
			fbModbusManager.addRequest_Write_Priority(WriteRequest := stModWrite_MotorSpeed);
			fbTON_WaitForMsg(IN := FALSE);
			eSMState := FINISH;
		END_IF
		
	FINISH:
		fbTON_WaitForMsg(IN := TRUE);
		
		IF fbTON_WaitForMsg.Q THEN
			fbModbusManager.addRequest_Read_Priority(ReadRequest := ADR(stModRead_Timeout));	
			fbTON_WaitForMsg(IN := FALSE);
		END_IF
		
		IF stModRead_Timeout.ReadRegsVals[1] = 0 THEN
			eSMState := WAIT;
			bBusy := FALSE;
			eState := E_DeviceState.IDLE;
			bInitialDose := FALSE;
		ELSE
			nRetries := nRetries + 1;
			IF nRetries > 5 THEN
				raiseAlarm(Priority := E_AlarmPriority.High, Label := 'Motor Counter Failed to Reach 0 After 5 Retries', Enabled := TRUE, DeviceAlarmID := 2);
				nRetries := 0;
				bBusy := FALSE;
				eSMState := WAIT;
				eState := E_DeviceState.IDLE;
				bInitialDose := FALSE;	
			END_IF
		END_IF

END_CASE

{warning 'add method implementation '}
METHOD executeDose : BOOL
VAR_INPUT
	DoseQtyMls: LREAL;
	DoseRateMlph: UINT;
	RequestComplete: 	POINTER TO BOOL;
END_VAR
VAR_OUTPUT
	RequestAccepted: BOOL;
END_VAR
(* setDose dispenses the amount requested at a user requested dose rate *)

IF ((bEnable AND bEnableComms) OR (eMode = E_DeviceMode.MANUAL)) AND ( NOT bInitialDose)  THEN
	
		nPumpSpeed_Requested := 40;
		tTimeToDose := REAL_TO_TIME(( ABS(DoseQtyMls) / (480.0*(UINT_TO_REAL(nPumpSpeed_Requested)/100.0))) * 60.0 *1000.0);  // Agrowtek maximum flow rate is 480 ml/min
		fbTONdoseTime.PT := tTimeToDose;
	
		IF tTimeToDose >= T#1S THEN
			nTimeToDoseSeconds := (TIME_TO_INT(tTimeToDose)/1000);
			nDoseQtyMls := nTimeToDoseSeconds * ((nPumpSpeed_Requested/100.0) * (480.0/60.0));
			eSMState := SET_TIME;
			eState := E_Devicestate.RUNNING;
			bBusy := TRUE;	
		END_IF
	END_IF
END_METHOD

METHOD FB_init : BOOL


VAR_INPUT
	bInitRetains : BOOL; // if TRUE, the retain variables are initialized (warm start / cold start)
	bInCopyCode : BOOL;  // if TRUE, the instance afterwards gets moved into the copy code (online change)
	
	PumpID: STRING;
	PumpDescription: STRING;
	PumpType: E_DosingPump;
	ManifoldModbusID: UINT; 
	
END_VAR
sID := PumpID;
sDescr := PumpDescription;
ePumpType := PumpType;
nModbusUnitID := ManifoldModbusID;
END_METHOD

METHOD getAdrMotorTime : UINT
VAR_INPUT
	PumpType: E_DosingPump;
END_VAR
// This method retrieves the Modbus register for the individual Agrowtek pump
// We need to do this because 5 pumps share the same Modbus slave ID, however have differing registers to write to

CASE PumpType OF
	
	E_DosingPump.PH_DOWN:
		getAdrReadWriteSpeed := 200;
		
	E_DosingPump.NUTRIENT_A:
		getAdrReadWriteSpeed := 201;
		
	E_DosingPump.NUTRIENT_B:
		getAdrReadWriteSpeed := 202;
		
	E_DosingPump.NUTRIENT_C:
		getAdrReadWriteSpeed := 203;
		
	E_DosingPump.PH_UP:
		getAdrReadWriteSpeed := 204;
		
END_CASE
END_METHOD

METHOD getAdrReadAccumRunTime : UINT
VAR_INPUT
	PumpType: E_DosingPump;
END_VAR

VAR
	Address: UINT;
END_VAR
// This method retrieves the Modbus register for the individual Agrowtek pump
// We need to do this because 5 pumps share the same Modbus slave ID, however have differing registers to write to

CASE PumpType OF
	
	E_DosingPump.PH_DOWN:
		Address := 16#64;
		
	E_DosingPump.NUTRIENT_A:
		Address := 16#65;
		
	E_DosingPump.NUTRIENT_B:
		Address := 16#66;

	E_DosingPump.NUTRIENT_C:
		Address := 16#67;
		
	E_DosingPump.PH_UP:
		Address := 16#68;
		
END_CASE

getAdrReadAccumRunTime := Address;
END_METHOD

METHOD getAdrReadWriteSpeed : UINT
VAR_INPUT
	PumpType: E_DosingPump;
END_VAR
// This method retrieves the Modbus register for the individual Agrowtek pump
// We need to do this because 5 pumps share the same Modbus slave ID, however have differing registers to write to

CASE PumpType OF
	
	E_DosingPump.PH_DOWN:
		getAdrReadWriteSpeed := 16#64;
		
	E_DosingPump.NUTRIENT_A:
		getAdrReadWriteSpeed := 16#65;
		
	E_DosingPump.NUTRIENT_B:
		getAdrReadWriteSpeed := 16#66;
		
	E_DosingPump.NUTRIENT_C:
		getAdrReadWriteSpeed := 16#67;
		
	E_DosingPump.PH_UP:
		getAdrReadWriteSpeed := 16#68;
		
END_CASE
END_METHOD

METHOD init_ModbusRequests : BOOL
VAR_INPUT
END_VAR
stModRead_MotorSpeed.SlaveAddress := nModbusUnitID;			
stModRead_MotorSpeed.AdrFirstSlaveRegisterRead := getAdrReadWriteSpeed(PumpType := ePumpType);
stModRead_MotorSpeed.QtyWordsToRead := 1;				// The value is a 16-bit word
stModRead_MotorSpeed.bRequestAccepted := FALSE;
stModRead_MotorSpeed.bRequestCompleted := FALSE;
stModRead_MotorSpeed.ReadRegsVals := GVL.ModbusEmptyBuffer;

stModRead_MotorRunTime.SlaveAddress := nModbusUnitID;			
stModRead_MotorRunTime.AdrFirstSlaveRegisterRead := getAdrReadAccumRunTime(PumpType := ePumpType);
stModRead_MotorRunTime.QtyWordsToRead := 1;				// The value is a 32-bit word
stModRead_MotorRunTime.bRequestAccepted := FALSE;
stModRead_MotorRunTime.bRequestCompleted := FALSE;
stModRead_MotorRunTime.ReadRegsVals := GVL.ModbusEmptyBuffer;

stModWrite_Timeout.SlaveAddress := nModbusUnitID;
stModWrite_Timeout.AdrFirstSlaveRegisterWrite := getAdrMotorTime(PumpType := ePumpType);
stModWrite_Timeout.bRequestAccepted := FALSE;
stModWrite_Timeout.bRequestCompleted := FALSE;
stModWrite_Timeout.QtyWordsToWrite := 1;

stModRead_Timeout.SlaveAddress := nModbusUnitID;
stModRead_Timeout.AdrFirstSlaveRegisterRead := 200;
stModRead_Timeout.bRequestAccepted := FALSE;
stModRead_Timeout.bRequestCompleted := FALSE;
stModRead_Timeout.ReadRegsVals := GVL.ModbusEmptyBuffer;


stModWrite_MotorSpeed.SlaveAddress := nModbusUnitID;
stModWrite_MotorSpeed.AdrFirstSlaveRegisterWrite := getAdrMotorTime(PumpType := ePumpType);
stModWrite_MotorSpeed.bRequestAccepted := FALSE;
stModWrite_MotorSpeed.bRequestCompleted := FALSE;
stModWrite_MotorSpeed.QtyWordsToWrite := 1;

stModWrite_SetID.SlaveAddress := 254;
stModWrite_SetID.AdrFirstSlaveRegisterWrite := 0;
stModWrite_SetID.bRequestAccepted := FALSE;
stModWrite_SetID.bRequestCompleted := FALSE;
stModWrite_SetID.QtyWordsToWrite := 1;
END_METHOD

METHOD readSpeed : BOOL
VAR_INPUT
END_VAR
fbModbusManager.addRequest_Read_Priority(ReadRequest := ADR(stModRead_MotorSpeed));
END_METHOD

METHOD setDoseQTY_InitDose : BOOL
VAR_INPUT
	DoseQtyMls: INT;
END_VAR

nDoseQtyMls := DoseQtyMls;
bInitialDose := TRUE;
END_METHOD

METHOD setModID : BOOL
VAR_INPUT
	DesiredID: UINT;
END_VAR
stModWrite_SetID.WriteRegVals[1] := DesiredID;
fbModbusManager.addRequest_Write_Priority(WriteRequest := ADR(stModWrite_SetID));
END_METHOD

METHOD setOFF : BOOL
VAR_INPUT
	RequestComplete: 	POINTER TO BOOL;
END_VAR
VAR_OUTPUT
	RequestAccepted: 	BOOL;
END_VAR
eSMState := DOSING_OFF_TRIG;
END_METHOD

METHOD setON : BOOL
VAR_INPUT
	RateMlph	 : 		UINT;
	RequestComplete: 	POINTER TO BOOL;
END_VAR

VAR_OUTPUT
	RequestAccepted: 	BOOL;
END_VAR
END_METHOD

METHOD setSpeed99 : BOOL
VAR_INPUT
END_VAR
nPumpSpeed_Requested := 99;
stModWrite_MotorSpeed.WriteRegVals[1] := UINT_TO_WORD(nPumpSpeed_Requested);
fbModbusManager.addRequest_Write_Priority(WriteRequest := ADR(stModWrite_MotorSpeed));
END_METHOD

END_FUNCTION_BLOCK

// ---- POUs/01 Actuators/Dosing Machine/FB_DosingPumpPRISMA.TcPOU
{attribute 'OPC.UA.DA.StructuredType' := '1'}
FUNCTION_BLOCK FB_DosingPumpPRISMA EXTENDS FB_BaseDevice IMPLEMENTS I_PumpDosing, I_Device

VAR_IN_OUT
	{attribute 'OPC.UA.DA' := '0'}
	fbModbusMaster: FB_ModbusMaster;
END_VAR

VAR
	// Modbus Variables\
	{attribute 'OPC.UA.DA' := '1'}
	{attribute 'OPC.UA.DA.Access' := '1'}
	nPumpID: UINT;	
	{attribute 'OPC.UA.DA' := '1'}
	{attribute 'OPC.UA.DA.Access' := '1'}
	nModbusUnitID: UINT; 
	
	//Pump Calibration / Capacity
	{attribute 'OPC.UA.DA' := '1'}
	{attribute 'OPC.UA.DA.Access' := '1'}
	nPumpCapacity: UINT;
	
	// 
	{attribute 'OPC.UA.DA' := '1'}
	nMaxRetries: UINT := 5;
	{attribute 'OPC.UA.DA' := '1'}
	nNumRetries: UINT := 0;
	
	{attribute 'OPC.UA.DA' := '0'}
	nReadRegsVals: ARRAY[1..10] OF WORD;
	{attribute 'OPC.UA.DA' := '0'}
	nWriteRegsVals: ARRAY[1..10] OF WORD;
	{attribute 'OPC.UA.DA' := '0'}
	nQtyWordsWrite: UINT;
	{attribute 'OPC.UA.DA' := '0'}
	nAddrWrite: UINT := 1;
	{attribute 'OPC.UA.DA' := '0'}
	nRegisterWordstoRead: UINT;
	{attribute 'OPC.UA.DA' := '0'}
	nAddrRead: UINT;
	
	// Async Statemachine Variables
	{attribute 'OPC.UA.DA' := '0'} 
	eSMState: (WAIT, READ_TRIG, READ, WRITE_TRIG, WRITE, SET_DOSE_TRIG, SET_DOSE, DOSE_ON_TRIG, DOSE_ON, DOSE_OFF_TRIG, DOSE_OFF, SET_BATCH_QTY_TRIG, SET_BATCH_QTY, SET_BATCH_TRIG, SET_BATCH, ERROR) := WAIT;
	{attribute 'OPC.UA.DA' := '0'} 
	bRequestFinished: POINTER TO BOOL;
	{attribute 'OPC.UA.DA' := '0'} 
	bRequestSentToMaster: BOOL 	:= FALSE;
	{attribute 'OPC.UA.DA' := '0'} 
	bRequestCompleted: BOOL 	:= FALSE;
	
	// Dosing Variables
	fbTONdoseTime: TON; // time the pump shall remain on at the nominated dosing rate
	{attribute 'OPC.UA.DA' := '0'}   
	fbTONdoseMsgDelay: TON := (PT := T#1000MS); // ensures pump has sufficient time to respond to request
	
	nDoseRateMLph: UINT;
	nDoseQtyMls: UINT;
	tTimeToDose: TIME;
	
	// Batch Dosing Variables
	bBatchPulse AT %Q*: BOOL := FALSE;
	nBatchQtyMl: UINT := 0;
	{attribute 'OPC.UA.DA' := '0'}   
	fbTONBatchMsgDelay: TON := (PT := T#100MS); // this gives time for the pump to be ready to receive a message
	
	
	(*
	  					SIMULATTION VARIABLES               
	*)	
	
END_VAR

fbTONdoseTime();
fbTONdoseMsgDelay();
fbTONBatchMsgDelay();

IF GVL.bAutoUpdateDeviceState THEN
	eState := eStateTarget;	
END_IF


IF eMode <> E_DeviceMode.SIMULATION THEN

	CASE eSMState OF
	
		WAIT :
		// Wait for eSMState to be changed in a method call
		nNumRetries := 0;
	
		READ_TRIG : 
			fbModbusMaster.readRegs(
				ReadRegsVals:= ADR(nReadRegsVals), 
				SlaveAddress:= nModbusUnitID, 
				QtyWordsToRead:= nRegisterWordstoRead, 
				AdrFirstSlaveRegisterRead:= nAddrRead, 
				bRequestCompleted:= ADR(bRequestCompleted), 
				bRequestAccepted=> bRequestSentToMaster);
				
			IF bRequestSentToMaster THEN
				eSMState := READ;
			END_IF
			
		
		READ :
			IF bRequestCompleted THEN	
				eSMState := WAIT; 						
				bRequestSentToMaster := FALSE;
				bRequestCompleted := TRUE;
				bBusy := FALSE;
			END_IF
		
			
		WRITE_TRIG :
			
			(*
			fbModbusMaster^.writeRegs(
				WriteRegVals:= nWriteRegsVals, 
				SlaveAddress:= nModbusUnitID, 
				QtyWordsToWrite:= nQtyWordsWrite, 
				AdrFirstSlaveRegisterWrite:= nAddrWrite, 
				bRequestCompleted:= ADR(bRequestCompleted), 
				bRequestAccepted=> bRequestSentToMaster);
				
				*)
			fbModbusMaster.writeReg(
				WriteRegVal:= nWriteRegsVals[1], 
				SlaveAddress:= nModbusUnitID, 
				AdrFirstSlaveRegisterWrite:= nAddrWrite, 
				bRequestCompleted:= ADR(bRequestCompleted), 
				bRequestAccepted=> bRequestSentToMaster);
				
			IF bRequestSentToMaster THEN  //Only progress if the ModbusMaster FB accepts the request - otherwise keep trying
				eSMState := WRITE;
			END_IF
			
		
		WRITE:
			IF bRequestCompleted THEN
				eSMState := WAIT;
				bRequestCompleted := FALSE;
				bRequestSentToMaster := FALSE;
				bBusy := FALSE;
			END_IF
			
		
		
		SET_DOSE_TRIG:
			
			IF bRequestSentToMaster = FALSE THEN
				IF fbModbusMaster.isBusy() = FALSE THEN
					nWriteRegsVals[1] := UINT_TO_WORD(nDoseRateMLph); 
					
					fbModbusMaster.writeRegs(
						WriteRegVals:= nWriteRegsVals, 
						SlaveAddress:= nModbusUnitID, 
						QtyWordsToWrite:= 1, 				
						AdrFirstSlaveRegisterWrite:= 16#94, 
						bRequestCompleted:= ADR(bRequestCompleted), 
						bRequestAccepted=> bRequestSentToMaster);
				END_IF
				
			ELSIF bRequestSentToMaster THEN	
				eSMState := SET_DOSE;
				bBusy := TRUE;
			END_IF	
			
			
		
		SET_DOSE:
			IF bRequestCompleted  THEN
				eSMState := DOSE_ON_TRIG;
				bRequestCompleted := FALSE;
				bRequestSentToMaster := FALSE;
				fbTONdoseMsgDelay(IN:= TRUE);		// give the pump 1s to respond	 
			END_IF	
		
		
		DOSE_ON_TRIG:
		
			IF bRequestSentToMaster = FALSE  THEN
				IF fbModbusMaster.isBusy() = FALSE THEN
					IF fbTONdoseMsgDelay.Q THEN
				
						nWriteRegsVals[1] := 16#01;
						
						fbModbusMaster.writeRegs(
							WriteRegVals:= nWriteRegsVals, 
							SlaveAddress:= nModbusUnitID, 
							QtyWordsToWrite:= 1, 				
							AdrFirstSlaveRegisterWrite:= 16#8C, 
							bRequestCompleted:= ADR(bRequestCompleted), 
							bRequestAccepted=> bRequestSentToMaster);
					END_IF
				END_IF
			ELSIF bRequestSentToMaster THEN
				eSMState := DOSE_ON;
				fbTONdoseMsgDelay.IN := FALSE;
				fbTONdoseTime(IN:= TRUE, PT := tTimeToDose); 
			END_IF
				
		DOSE_ON:
			IF bRequestCompleted THEN
				eSMState := DOSE_OFF_TRIG;
				bRequestCompleted := FALSE;
				bRequestSentToMaster := FALSE;
			END_IF
			
	
		DOSE_OFF_TRIG:
			
			IF bRequestSentToMaster = FALSE THEN
				IF fbModbusMaster.isBusy() = FALSE THEN
					IF fbTONdoseTime.Q THEN
						nWriteRegsVals[1] := 16#0;
						fbModbusMaster.writeRegs(
							WriteRegVals:= nWriteRegsVals, 
							SlaveAddress:= nModbusUnitID, 
							QtyWordsToWrite:= 1,  // 8 bytes from 40141 to 40149
							AdrFirstSlaveRegisterWrite:= 16#8C, 
							bRequestCompleted:= ADR(bRequestCompleted), 
							bRequestAccepted=> bRequestSentToMaster);
					END_IF
				END_IF
			ELSIF bRequestSentToMaster THEN
				eSMState := DOSE_OFF;
			END_IF
				
		DOSE_OFF:
			IF bRequestCompleted  AND fbModbusMaster.Error() = FALSE THEN
				eSMState := WAIT;
				bRequestCompleted := FALSE;
				bRequestSentToMaster := FALSE;
				bBusy := FALSE;
				fbTONdoseTime.IN := FALSE;
				bRequestFinished^ := TRUE;
				nDoseQtyMls := 0;  // Set this to zero so that the historised tag can capture duplicate successive doses
			END_IF
			
			IF fbModbusMaster.Error() = TRUE THEN
				eSMState := SET_DOSE_TRIG;
				nNumRetries := nNumRetries + 1;
			END_IF
			
			IF nNumRetries > nMaxRetries THEN
				//Raise an error event for modbus communications
			END_IF
			
			
		SET_BATCH_QTY_TRIG:
			IF bRequestSentToMaster = FALSE THEN
				IF fbModbusMaster.isBusy() = FALSE THEN
					
					nWriteRegsVals[1] := UINT_TO_WORD(nDoseQtyMls); 
					fbModbusMaster.writeRegs(
						WriteRegVals:= nWriteRegsVals, 
						SlaveAddress:= nModbusUnitID, 
						QtyWordsToWrite:= 1, 				
						AdrFirstSlaveRegisterWrite:= 16#DA, 
						bRequestCompleted:= ADR(bRequestCompleted), 
						bRequestAccepted=> bRequestSentToMaster);
				END_IF
			ELSIF bRequestSentToMaster THEN	
				eSMState := SET_BATCH_QTY;
			END_IF
	
		SET_BATCH_QTY:
			IF bRequestCompleted  THEN
				bRequestCompleted := FALSE;
				bRequestSentToMaster := FALSE;
				fbTONBatchMsgDelay(IN := TRUE);
				eSMState := SET_BATCH_TRIG;
			END_IF	
				
		SET_BATCH_TRIG:
			IF fbTONBatchMsgDelay.Q = TRUE THEN
				bBatchPulse := TRUE;
				fbTONBatchMsgDelay(IN := FALSE);
				fbTONBatchMsgDelay(IN := TRUE);
				eSMState := SET_BATCH;
			END_IF
			
		SET_BATCH:
			IF fbTONBatchMsgDelay.Q = TRUE AND fbModbusMaster.Error() = FALSE THEN
				bBatchPulse := FALSE;			
				fbTONBatchMsgDelay.IN := FALSE;
				bBusy := FALSE;
				bRequestCompleted := FALSE;
				bRequestSentToMaster := FALSE;
				eSMState := WAIT;
			END_IF
			
			IF fbModbusMaster.Error() = TRUE THEN
				eSMState := SET_DOSE_TRIG;
				nNumRetries := nNumRetries + 1;
			END_IF
			
			IF nNumRetries > nMaxRetries THEN
				//Raise an error event for modbus communications
			END_IF
		END_CASE
	
	(*
					SIMULATION CODE
	*)
	
	ELSIF eMode = E_DeviceMode.SIMULATION THEN
		
		IF eSMState = SET_DOSE_TRIG THEN  					// we are not at our desired state
			
